// TIA Portal V15.1 export
// export: Created 2024-05-17T05:38:33.8668147Z, ExportSetting WithDefaults, DisplayName Totally Integrated Automation Portal, DisplayVersion V15.1 Update 5, DisplayName TIA Portal Openness, DisplayVersion V15.1 Update 5, DisplayName SINAMICS Startdrive Advanced, DisplayVersion V15.1, DisplayName G130, G150, S120, S150, SINAMICS MV, S210, DisplayVersion V15.1, DisplayName G110M, G120, G120C, G120D, G120P, DisplayVersion V15.1, DisplayName STEP 7 Professional, DisplayVersion V15.1 Update 5, DisplayName STEP 7 Safety, DisplayVersion V15.1, DisplayName WinCC Professional, DisplayVersion V15.1 Update 5, DisplayName SIMATIC Visualization Architect, DisplayVersion V15.1
FUNCTION_BLOCK "LProcSel5SPResFreq"   // FB1733, FBD
TITLE = LProcSel5SPResFreq
{ S7_Optimized_Access := 'FALSE' }
AUTHOR : VCC
FAMILY : ProcEq
NAME : Sel5SP
VERSION : 0.1
// ================================================================================
// This makes the selection of one set-point among 5 in function of the production 
// modes.
// The selection is made via a set-point request integer from 1 to 5.
// An external value is possible to be selected to set-point 1.
// It includes also 5 set-points to reject resonance frequencies if there are.
// ================================================================================
// stored: AutoNumber false, IsIECCheckEnabled false, SetENOAutomatically False, UDAEnableTagReadback false
   VAR_INPUT
      I_ExtSP1_Value { ExternalAccessible := 'False'; ExternalVisible := 'False'; ExternalWritable := 'False'} : Real;   // External Set-point 1
      H_Normalbandwidthmode { ExternalAccessible := 'False'; ExternalVisible := 'False'; ExternalWritable := 'False'} : Bool := TRUE;   // Each resonance frequency his own bandwidth
      H_SPResonance1 : Real;   // Set-point 1 Resonance frequency
      H_SPResonance2 : Real;   // Set-point 2 Resonance frequency
      H_SPResonance3 : Real;   // Set-point 3 Resonance frequency
      H_SPResonance4 : Real;   // Set-point 4 Resonance frequency
      H_SPBandwidth1 : Real;   // Set-point 1 Bandwidth (for resonance frequency)
      H_SPBandwidth2 : Real;   // Set-point 2 Bandwidth (for resonance frequency)
      H_SPBandwidth3 : Real;   // Set-point 3 Bandwidth (for resonance frequency)
      H_SPBandwidth4 : Real;   // Set-point 4 Bandwidth (for resonance frequency)
      I_SPReq : Int;   // Index Set-point Request
      I_ExtSP1 : Bool;   // External Set-point 1 Request
   END_VAR
   VAR_OUTPUT
      O_SPSel : Real;   // Set-point selected
      H_Anim : Word;   // HMI Animation word
   END_VAR
   VAR_IN_OUT
      H_SetpntAllowed : Bool := TRUE;   // Setpoint is OK and allowed
      H_SP1 : Real;   // Set-point 1
      H_SP2 : Real;   // Set-point 2
      H_SP3 : Real;   // Set-point 3
      H_SP4 : Real;   // Set-point 4
      H_SP5 : Real;   // Set-point 5
   END_VAR
   VAR DB_SPECIFIC
      RunNormalOnce { ExternalAccessible := 'False'; ExternalVisible := 'False'; ExternalWritable := 'False'} : Bool := TRUE;   // Check all frequences once - mode is changed
      RunNotNormalOnce { ExternalAccessible := 'False'; ExternalVisible := 'False'; ExternalWritable := 'False'} : Bool;   // Check all frequences once - mode is changed
      SetpntChanged { ExternalAccessible := 'False'; ExternalVisible := 'False'; ExternalWritable := 'False'} : Bool;   // Setpoint is changed
      SetpntResChanged { ExternalAccessible := 'False'; ExternalVisible := 'False'; ExternalWritable := 'False'} : Bool;   // Setpoint Resonance frequency is changed
      SetpntBwdChanged { ExternalAccessible := 'False'; ExternalVisible := 'False'; ExternalWritable := 'False'} : Bool;   // Setpoint bandwidth is changed
      CheckResSetpoints { ExternalAccessible := 'False'; ExternalVisible := 'False'; ExternalWritable := 'False'} : Bool;   // Check all frequences because mode is changed
      ClrGreatestbandwidth { ExternalAccessible := 'False'; ExternalVisible := 'False'; ExternalWritable := 'False'} : Bool;   // Clear greatest bandwidth to search new value
      Greatestbandwidth { ExternalAccessible := 'False'; ExternalVisible := 'False'; ExternalWritable := 'False'} : Real;   // Greatest bandwidth from those who where entered
      MinResSetp1 { ExternalAccessible := 'False'; ExternalVisible := 'False'; ExternalWritable := 'False'} : Real;   // Calculated min. res. Setpoint 1
      MaxResSetp1 { ExternalAccessible := 'False'; ExternalVisible := 'False'; ExternalWritable := 'False'} : Real;   // Calculated max. res. Setpoint 1
      MinResSetp2 { ExternalAccessible := 'False'; ExternalVisible := 'False'; ExternalWritable := 'False'} : Real;   // Calculated min. res. Setpoint 2
      MaxResSetp2 { ExternalAccessible := 'False'; ExternalVisible := 'False'; ExternalWritable := 'False'} : Real;   // Calculated max. res. Setpoint 2
      MinResSetp3 { ExternalAccessible := 'False'; ExternalVisible := 'False'; ExternalWritable := 'False'} : Real;   // Calculated min. res. Setpoint 3
      MaxResSetp3 { ExternalAccessible := 'False'; ExternalVisible := 'False'; ExternalWritable := 'False'} : Real;   // Calculated max. res. Setpoint 3
      MinResSetp4 { ExternalAccessible := 'False'; ExternalVisible := 'False'; ExternalWritable := 'False'} : Real;   // Calculated min. res. Setpoint 4
      MaxResSetp4 { ExternalAccessible := 'False'; ExternalVisible := 'False'; ExternalWritable := 'False'} : Real;   // Calculated max. res. Setpoint 4
      S_NormalBndWdth { ExternalAccessible := 'False'; ExternalVisible := 'False'; ExternalWritable := 'False'} : Bool;   // Step Normal Bandwidth
      S_NoNormalBndWdth { ExternalAccessible := 'False'; ExternalVisible := 'False'; ExternalWritable := 'False'} : Bool;   // Step No Normal Bandwidth
      SPOld1 { ExternalAccessible := 'False'; ExternalVisible := 'False'; ExternalWritable := 'False'} : Real;   // Set-point 1
      SPOld2 { ExternalAccessible := 'False'; ExternalVisible := 'False'; ExternalWritable := 'False'} : Real;   // Set-point 2
      SPOld3 { ExternalAccessible := 'False'; ExternalVisible := 'False'; ExternalWritable := 'False'} : Real;   // Set-point 3
      SPOld4 { ExternalAccessible := 'False'; ExternalVisible := 'False'; ExternalWritable := 'False'} : Real;   // Set-point 4
      SPOld5 { ExternalAccessible := 'False'; ExternalVisible := 'False'; ExternalWritable := 'False'} : Real;   // Set-point 5
      SPResonanceOld1 { ExternalAccessible := 'False'; ExternalVisible := 'False'; ExternalWritable := 'False'} : Real;   // Set-point 1 Resonance frequency
      SPResonanceOld2 { ExternalAccessible := 'False'; ExternalVisible := 'False'; ExternalWritable := 'False'} : Real;   // Set-point 2 Resonance frequency
      SPResonanceOld3 { ExternalAccessible := 'False'; ExternalVisible := 'False'; ExternalWritable := 'False'} : Real;   // Set-point 3 Resonance frequency
      SPResonanceOld4 { ExternalAccessible := 'False'; ExternalVisible := 'False'; ExternalWritable := 'False'} : Real;   // Set-point 4 Resonance frequency
      SPBandwidthOld1 { ExternalAccessible := 'False'; ExternalVisible := 'False'; ExternalWritable := 'False'} : Real;   // Set-point 1 Bandwidth (for resonance frequency)
      SPBandwidthOld2 { ExternalAccessible := 'False'; ExternalVisible := 'False'; ExternalWritable := 'False'} : Real;   // Set-point 2 Bandwidth (for resonance frequency)
      SPBandwidthOld3 { ExternalAccessible := 'False'; ExternalVisible := 'False'; ExternalWritable := 'False'} : Real;   // Set-point 3 Bandwidth (for resonance frequency)
      SPBandwidthOld4 { ExternalAccessible := 'False'; ExternalVisible := 'False'; ExternalWritable := 'False'} : Real;   // Set-point 4 Bandwidth (for resonance frequency)
   END_VAR
   VAR_TEMP   // added for the SCL form of the ladder/FBD networks
      _w1 : Bool;
      _w2 : Bool;
      _w3 : Bool;
   END_VAR
BEGIN

REGION Network 1: **** 4.6 - Machine status - Indications **** Controller Animation word 1 for HMI
   // Controller Animation word 1 for HMI
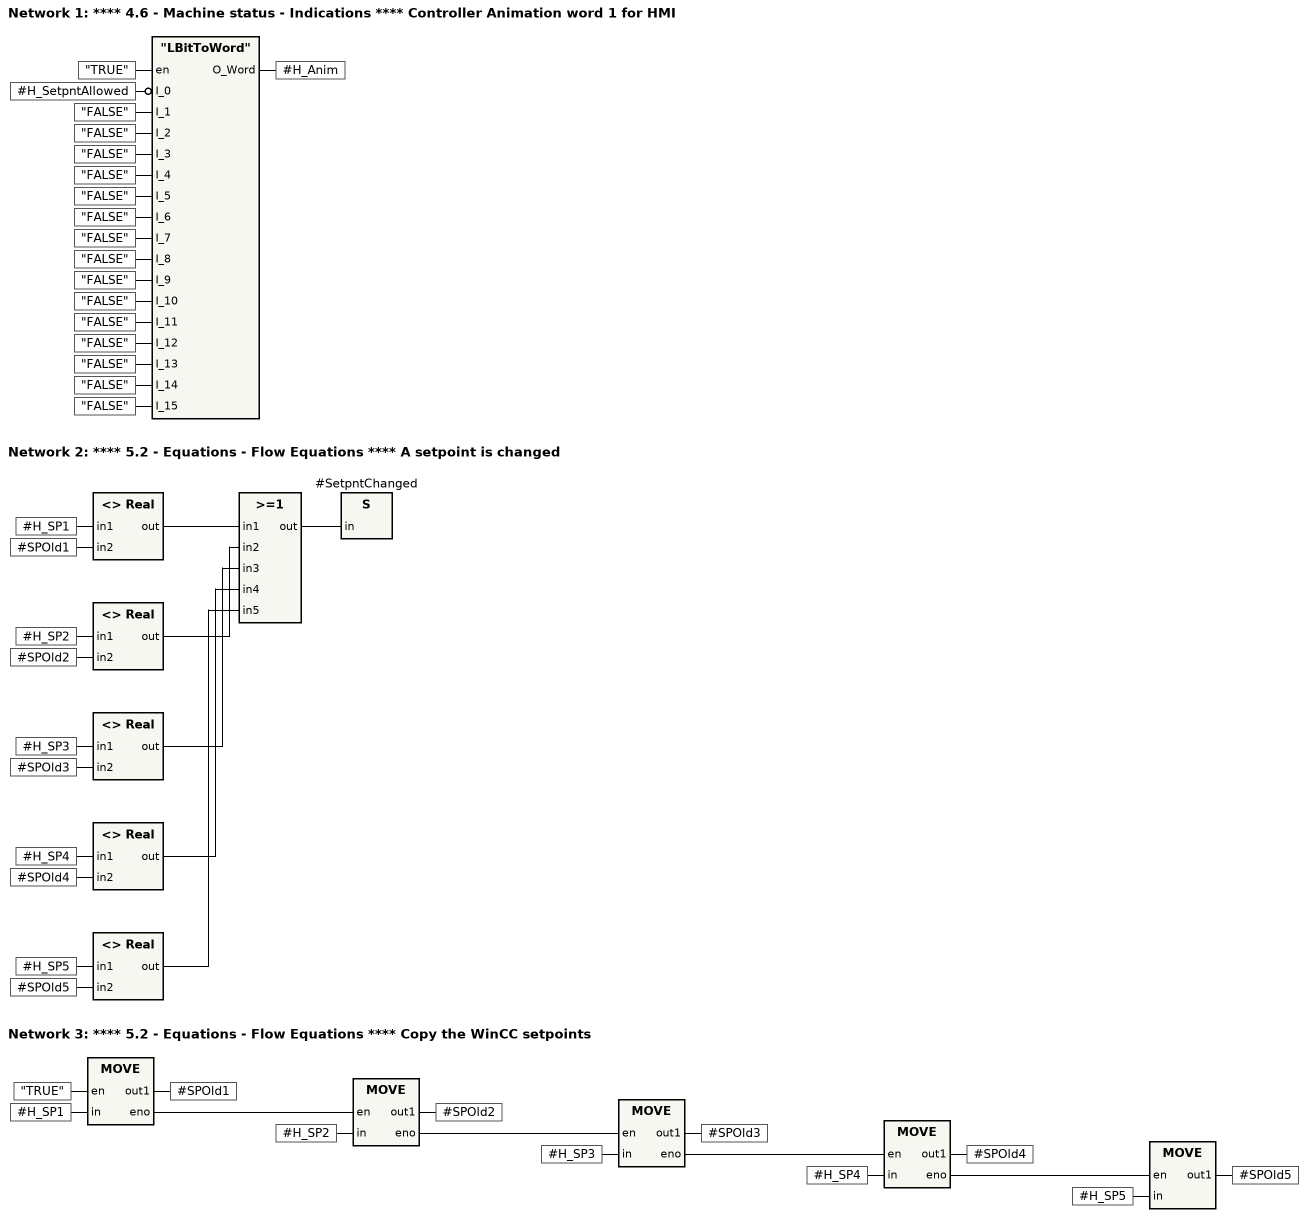
   IF "TRUE" THEN
       "LBitToWord"(I_0 := NOT #H_SetpntAllowed,
                    I_1 := "FALSE",
                    I_2 := "FALSE",
                    I_3 := "FALSE",
                    I_4 := "FALSE",
                    I_5 := "FALSE",
                    I_6 := "FALSE",
                    I_7 := "FALSE",
                    I_8 := "FALSE",
                    I_9 := "FALSE",
                    I_10 := "FALSE",
                    I_11 := "FALSE",
                    I_12 := "FALSE",
                    I_13 := "FALSE",
                    I_14 := "FALSE",
                    I_15 := "FALSE",
                    O_Word => #H_Anim);
   END_IF;
END_REGION

REGION Network 2: **** 5.2 - Equations - Flow Equations **** A setpoint is changed
   // A setpoint is changed
   IF (#H_SP1 <> #SPOld1) OR (#H_SP2 <> #SPOld2) OR (#H_SP3 <> #SPOld3) OR (#H_SP4 <> #SPOld4) OR (#H_SP5 <> #SPOld5) THEN
       #SetpntChanged := TRUE;
   END_IF;
END_REGION

REGION Network 3: **** 5.2 - Equations - Flow Equations **** Copy the WinCC setpoints
   // Copy the WinCC setpoints
   // ENO of a box is taken as its EN; it also drops when the box reports an error
   IF "TRUE" THEN
       #SPOld1 := #H_SP1;
       #SPOld2 := #H_SP2;
       #SPOld3 := #H_SP3;
       #SPOld4 := #H_SP4;
       #SPOld5 := #H_SP5;
   END_IF;
END_REGION

REGION Network 4: **** 5.2 - Equations - Flow Equations **** A setpoint of resonance is changed
   // A setpoint of resonance is changed
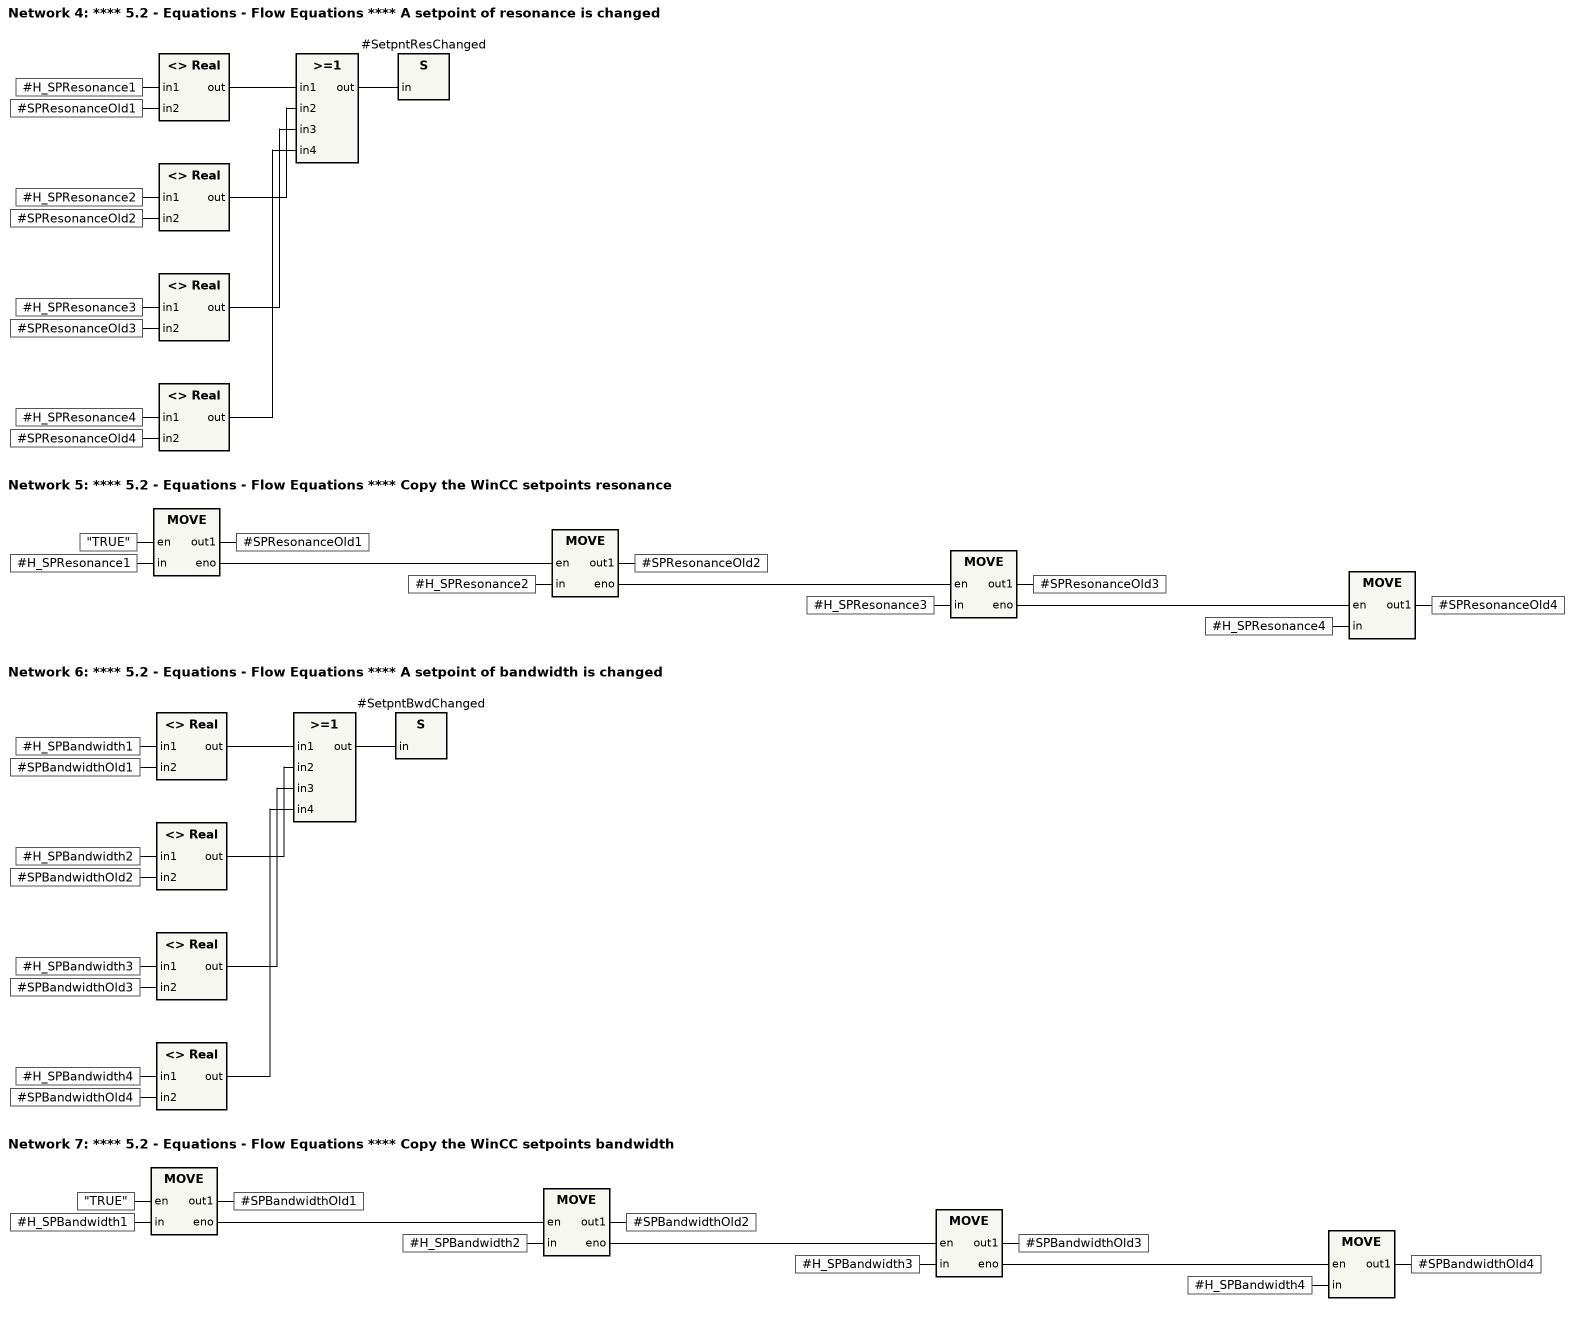
   IF (#H_SPResonance1 <> #SPResonanceOld1) OR (#H_SPResonance2 <> #SPResonanceOld2) OR (#H_SPResonance3 <> #SPResonanceOld3) OR (#H_SPResonance4 <> #SPResonanceOld4) THEN
       #SetpntResChanged := TRUE;
   END_IF;
END_REGION

REGION Network 5: **** 5.2 - Equations - Flow Equations **** Copy the WinCC setpoints resonance
   // Copy the WinCC setpoints resonance
   // ENO of a box is taken as its EN; it also drops when the box reports an error
   IF "TRUE" THEN
       #SPResonanceOld1 := #H_SPResonance1;
       #SPResonanceOld2 := #H_SPResonance2;
       #SPResonanceOld3 := #H_SPResonance3;
       #SPResonanceOld4 := #H_SPResonance4;
   END_IF;
END_REGION

REGION Network 6: **** 5.2 - Equations - Flow Equations **** A setpoint of bandwidth is changed
   // A setpoint of bandwidth is changed
   IF (#H_SPBandwidth1 <> #SPBandwidthOld1) OR (#H_SPBandwidth2 <> #SPBandwidthOld2) OR (#H_SPBandwidth3 <> #SPBandwidthOld3) OR (#H_SPBandwidth4 <> #SPBandwidthOld4) THEN
       #SetpntBwdChanged := TRUE;
   END_IF;
END_REGION

REGION Network 7: **** 5.2 - Equations - Flow Equations **** Copy the WinCC setpoints bandwidth
   // Copy the WinCC setpoints bandwidth
   // ENO of a box is taken as its EN; it also drops when the box reports an error
   IF "TRUE" THEN
       #SPBandwidthOld1 := #H_SPBandwidth1;
       #SPBandwidthOld2 := #H_SPBandwidth2;
       #SPBandwidthOld3 := #H_SPBandwidth3;
       #SPBandwidthOld4 := #H_SPBandwidth4;
   END_IF;
END_REGION

REGION Network 8: **** 5.2 - Equations - Flow Equations **** Selection Set-point 1
   // Selection Set-point 1
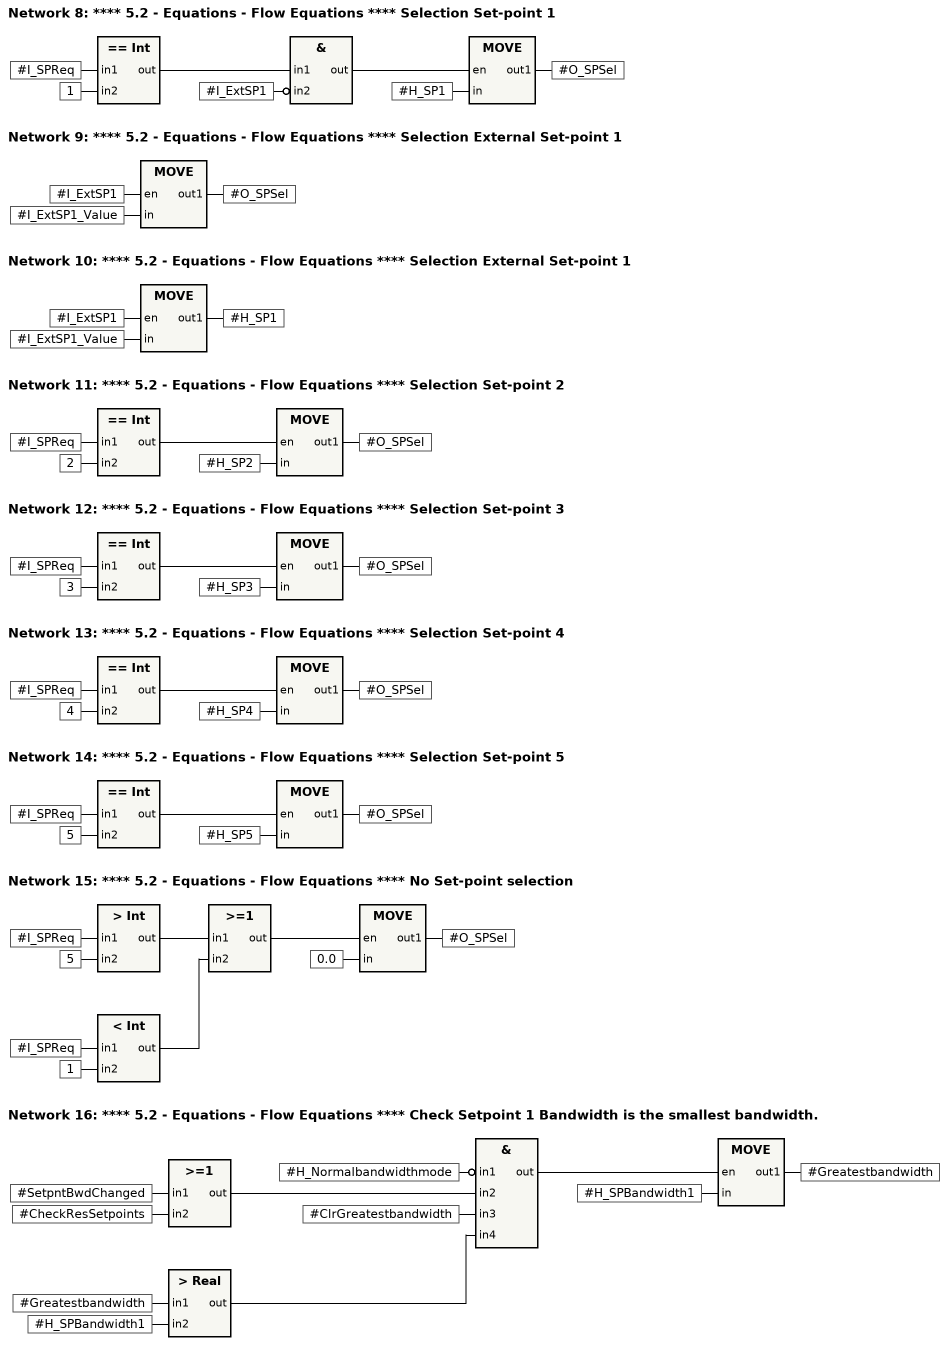
   IF (#I_SPReq = 1) AND NOT #I_ExtSP1 THEN #O_SPSel := #H_SP1; END_IF;
END_REGION

REGION Network 9: **** 5.2 - Equations - Flow Equations **** Selection External Set-point 1
   // Selection External Set-point 1
   IF #I_ExtSP1 THEN #O_SPSel := #I_ExtSP1_Value; END_IF;
END_REGION

REGION Network 10: **** 5.2 - Equations - Flow Equations **** Selection External Set-point 1
   // Selection External Set-point 1
   IF #I_ExtSP1 THEN #H_SP1 := #I_ExtSP1_Value; END_IF;
END_REGION

REGION Network 11: **** 5.2 - Equations - Flow Equations **** Selection Set-point 2
   // Selection Set-point 2
   IF #I_SPReq = 2 THEN #O_SPSel := #H_SP2; END_IF;
END_REGION

REGION Network 12: **** 5.2 - Equations - Flow Equations **** Selection Set-point 3
   // Selection Set-point 3
   IF #I_SPReq = 3 THEN #O_SPSel := #H_SP3; END_IF;
END_REGION

REGION Network 13: **** 5.2 - Equations - Flow Equations **** Selection Set-point 4
   // Selection Set-point 4
   IF #I_SPReq = 4 THEN #O_SPSel := #H_SP4; END_IF;
END_REGION

REGION Network 14: **** 5.2 - Equations - Flow Equations **** Selection Set-point 5
   // Selection Set-point 5
   IF #I_SPReq = 5 THEN #O_SPSel := #H_SP5; END_IF;
END_REGION

REGION Network 15: **** 5.2 - Equations - Flow Equations **** No Set-point selection
   // No Set-point selection
   IF (#I_SPReq > 5) OR (#I_SPReq < 1) THEN #O_SPSel := 0.0; END_IF;
END_REGION

REGION Network 16: **** 5.2 - Equations - Flow Equations **** Check Setpoint 1 Bandwidth is the smallest bandwidth.
   // Check Setpoint 1 Bandwidth is the smallest bandwidth.
   IF NOT #H_Normalbandwidthmode AND (#SetpntBwdChanged OR #CheckResSetpoints) AND #ClrGreatestbandwidth AND (#Greatestbandwidth > #H_SPBandwidth1) THEN
       #Greatestbandwidth := #H_SPBandwidth1;
   END_IF;
END_REGION

REGION Network 17: **** 5.2 - Equations - Flow Equations **** Check Setpoint 2 Bandwidth is the smallest bandwidth.
   // Check Setpoint 2 Bandwidth is the smallest bandwidth.
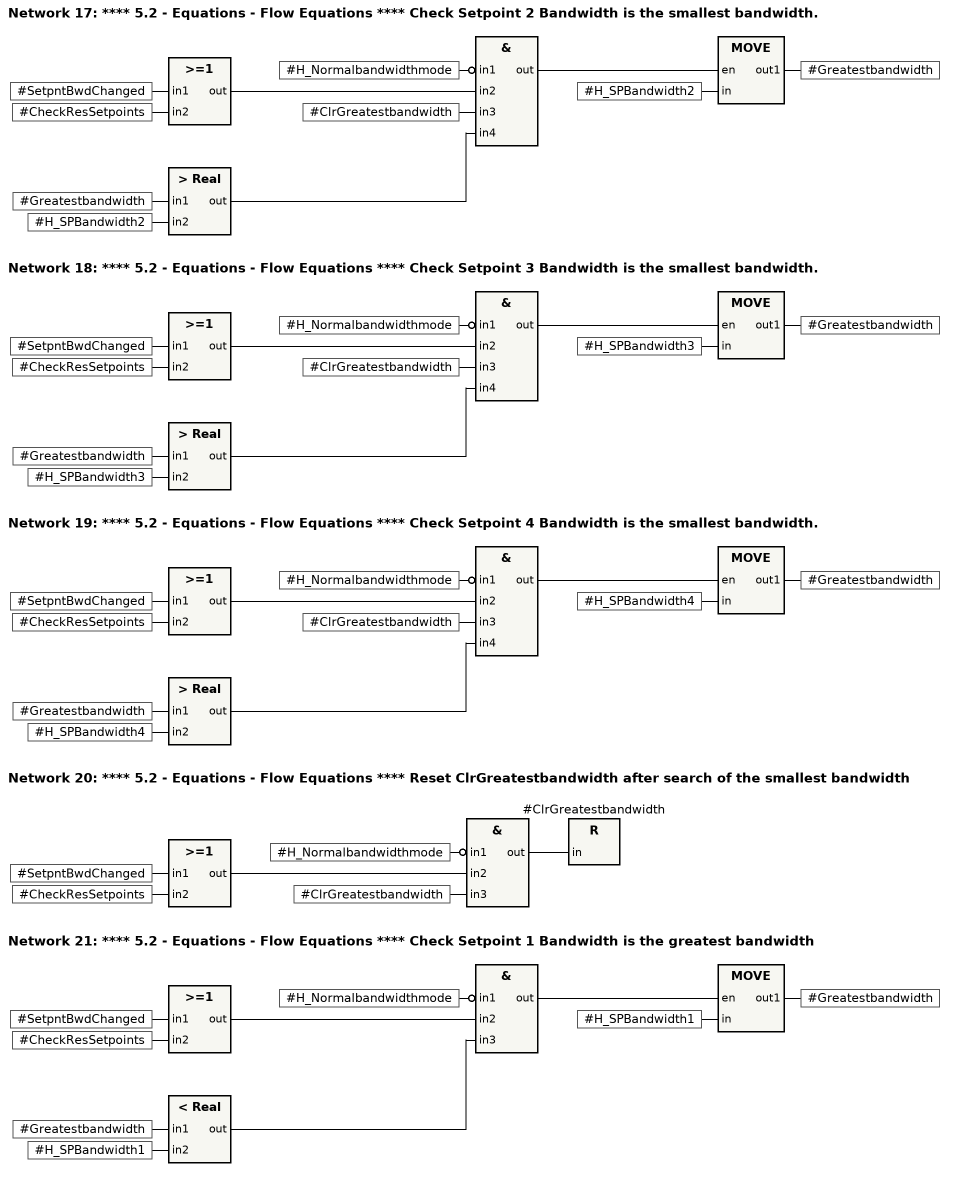
   IF NOT #H_Normalbandwidthmode AND (#SetpntBwdChanged OR #CheckResSetpoints) AND #ClrGreatestbandwidth AND (#Greatestbandwidth > #H_SPBandwidth2) THEN
       #Greatestbandwidth := #H_SPBandwidth2;
   END_IF;
END_REGION

REGION Network 18: **** 5.2 - Equations - Flow Equations **** Check Setpoint 3 Bandwidth is the smallest bandwidth.
   // Check Setpoint 3 Bandwidth is the smallest bandwidth.
   IF NOT #H_Normalbandwidthmode AND (#SetpntBwdChanged OR #CheckResSetpoints) AND #ClrGreatestbandwidth AND (#Greatestbandwidth > #H_SPBandwidth3) THEN
       #Greatestbandwidth := #H_SPBandwidth3;
   END_IF;
END_REGION

REGION Network 19: **** 5.2 - Equations - Flow Equations **** Check Setpoint 4 Bandwidth is the smallest bandwidth.
   // Check Setpoint 4 Bandwidth is the smallest bandwidth.
   IF NOT #H_Normalbandwidthmode AND (#SetpntBwdChanged OR #CheckResSetpoints) AND #ClrGreatestbandwidth AND (#Greatestbandwidth > #H_SPBandwidth4) THEN
       #Greatestbandwidth := #H_SPBandwidth4;
   END_IF;
END_REGION

REGION Network 20: **** 5.2 - Equations - Flow Equations **** Reset ClrGreatestbandwidth after search of the smallest bandwidth
   // Reset ClrGreatestbandwidth after search of the smallest bandwidth
   IF NOT #H_Normalbandwidthmode AND (#SetpntBwdChanged OR #CheckResSetpoints) AND #ClrGreatestbandwidth THEN
       #ClrGreatestbandwidth := FALSE;
   END_IF;
END_REGION

REGION Network 21: **** 5.2 - Equations - Flow Equations **** Check Setpoint 1 Bandwidth is the greatest bandwidth
   // Check Setpoint 1 Bandwidth is the greatest bandwidth
   IF NOT #H_Normalbandwidthmode AND (#SetpntBwdChanged OR #CheckResSetpoints) AND (#Greatestbandwidth < #H_SPBandwidth1) THEN
       #Greatestbandwidth := #H_SPBandwidth1;
   END_IF;
END_REGION

REGION Network 22: **** 5.2 - Equations - Flow Equations **** Check Setpoint 2 Bandwidth is the greatest bandwidth
   // Check Setpoint 2 Bandwidth is the greatest bandwidth
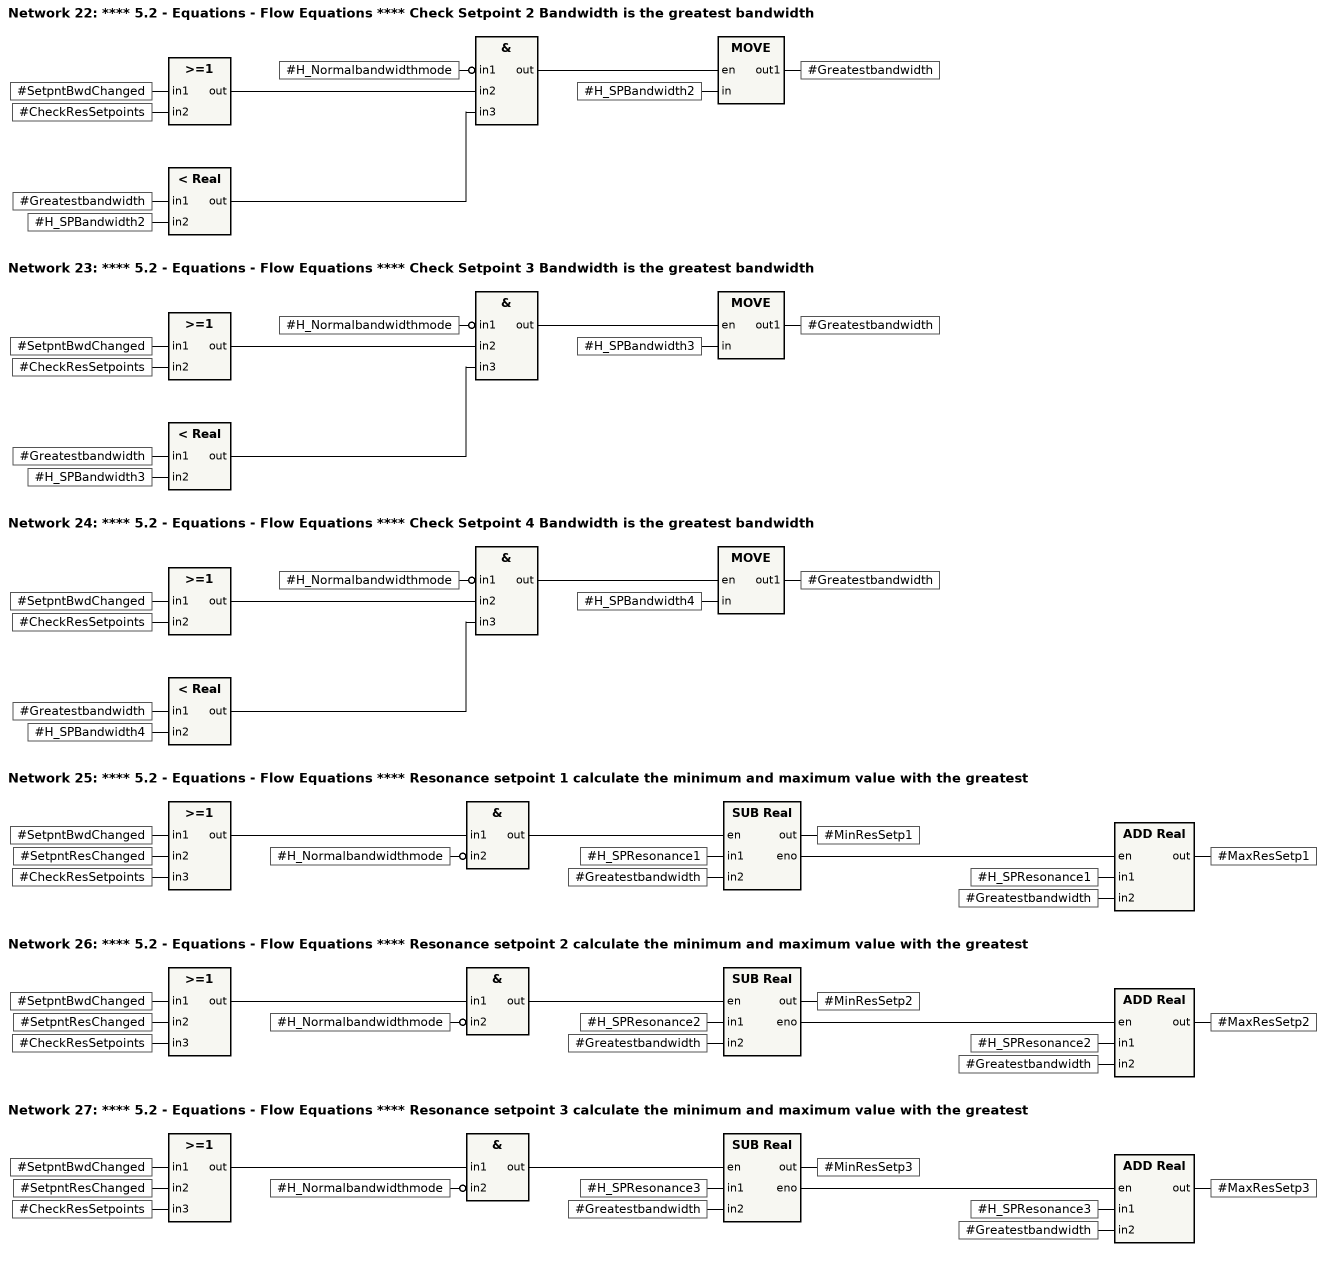
   IF NOT #H_Normalbandwidthmode AND (#SetpntBwdChanged OR #CheckResSetpoints) AND (#Greatestbandwidth < #H_SPBandwidth2) THEN
       #Greatestbandwidth := #H_SPBandwidth2;
   END_IF;
END_REGION

REGION Network 23: **** 5.2 - Equations - Flow Equations **** Check Setpoint 3 Bandwidth is the greatest bandwidth
   // Check Setpoint 3 Bandwidth is the greatest bandwidth
   IF NOT #H_Normalbandwidthmode AND (#SetpntBwdChanged OR #CheckResSetpoints) AND (#Greatestbandwidth < #H_SPBandwidth3) THEN
       #Greatestbandwidth := #H_SPBandwidth3;
   END_IF;
END_REGION

REGION Network 24: **** 5.2 - Equations - Flow Equations **** Check Setpoint 4 Bandwidth is the greatest bandwidth
   // Check Setpoint 4 Bandwidth is the greatest bandwidth
   IF NOT #H_Normalbandwidthmode AND (#SetpntBwdChanged OR #CheckResSetpoints) AND (#Greatestbandwidth < #H_SPBandwidth4) THEN
       #Greatestbandwidth := #H_SPBandwidth4;
   END_IF;
END_REGION

REGION Network 25: **** 5.2 - Equations - Flow Equations **** Resonance setpoint 1 calculate the minimum and maximum value with the greatest
   // Resonance setpoint 1 calculate the minimum and maximum value with the greatest 
   // bandwidth
   // ENO of a box is taken as its EN; it also drops when the box reports an error
   IF (#SetpntBwdChanged OR #SetpntResChanged OR #CheckResSetpoints) AND NOT #H_Normalbandwidthmode THEN
       #MinResSetp1 := #H_SPResonance1 - #Greatestbandwidth;
       #MaxResSetp1 := #H_SPResonance1 + #Greatestbandwidth;
   END_IF;
END_REGION

REGION Network 26: **** 5.2 - Equations - Flow Equations **** Resonance setpoint 2 calculate the minimum and maximum value with the greatest
   // Resonance setpoint 2 calculate the minimum and maximum value with the greatest 
   // bandwidth
   // ENO of a box is taken as its EN; it also drops when the box reports an error
   IF (#SetpntBwdChanged OR #SetpntResChanged OR #CheckResSetpoints) AND NOT #H_Normalbandwidthmode THEN
       #MinResSetp2 := #H_SPResonance2 - #Greatestbandwidth;
       #MaxResSetp2 := #H_SPResonance2 + #Greatestbandwidth;
   END_IF;
END_REGION

REGION Network 27: **** 5.2 - Equations - Flow Equations **** Resonance setpoint 3 calculate the minimum and maximum value with the greatest
   // Resonance setpoint 3 calculate the minimum and maximum value with the greatest 
   // bandwidth
   // ENO of a box is taken as its EN; it also drops when the box reports an error
   IF (#SetpntBwdChanged OR #SetpntResChanged OR #CheckResSetpoints) AND NOT #H_Normalbandwidthmode THEN
       #MinResSetp3 := #H_SPResonance3 - #Greatestbandwidth;
       #MaxResSetp3 := #H_SPResonance3 + #Greatestbandwidth;
   END_IF;
END_REGION

REGION Network 28: **** 5.2 - Equations - Flow Equations **** Resonance setpoint 4 calculate the minimum and maximum value with the greatest
   // Resonance setpoint 4 calculate the minimum and maximum value with the greatest 
   // bandwidth
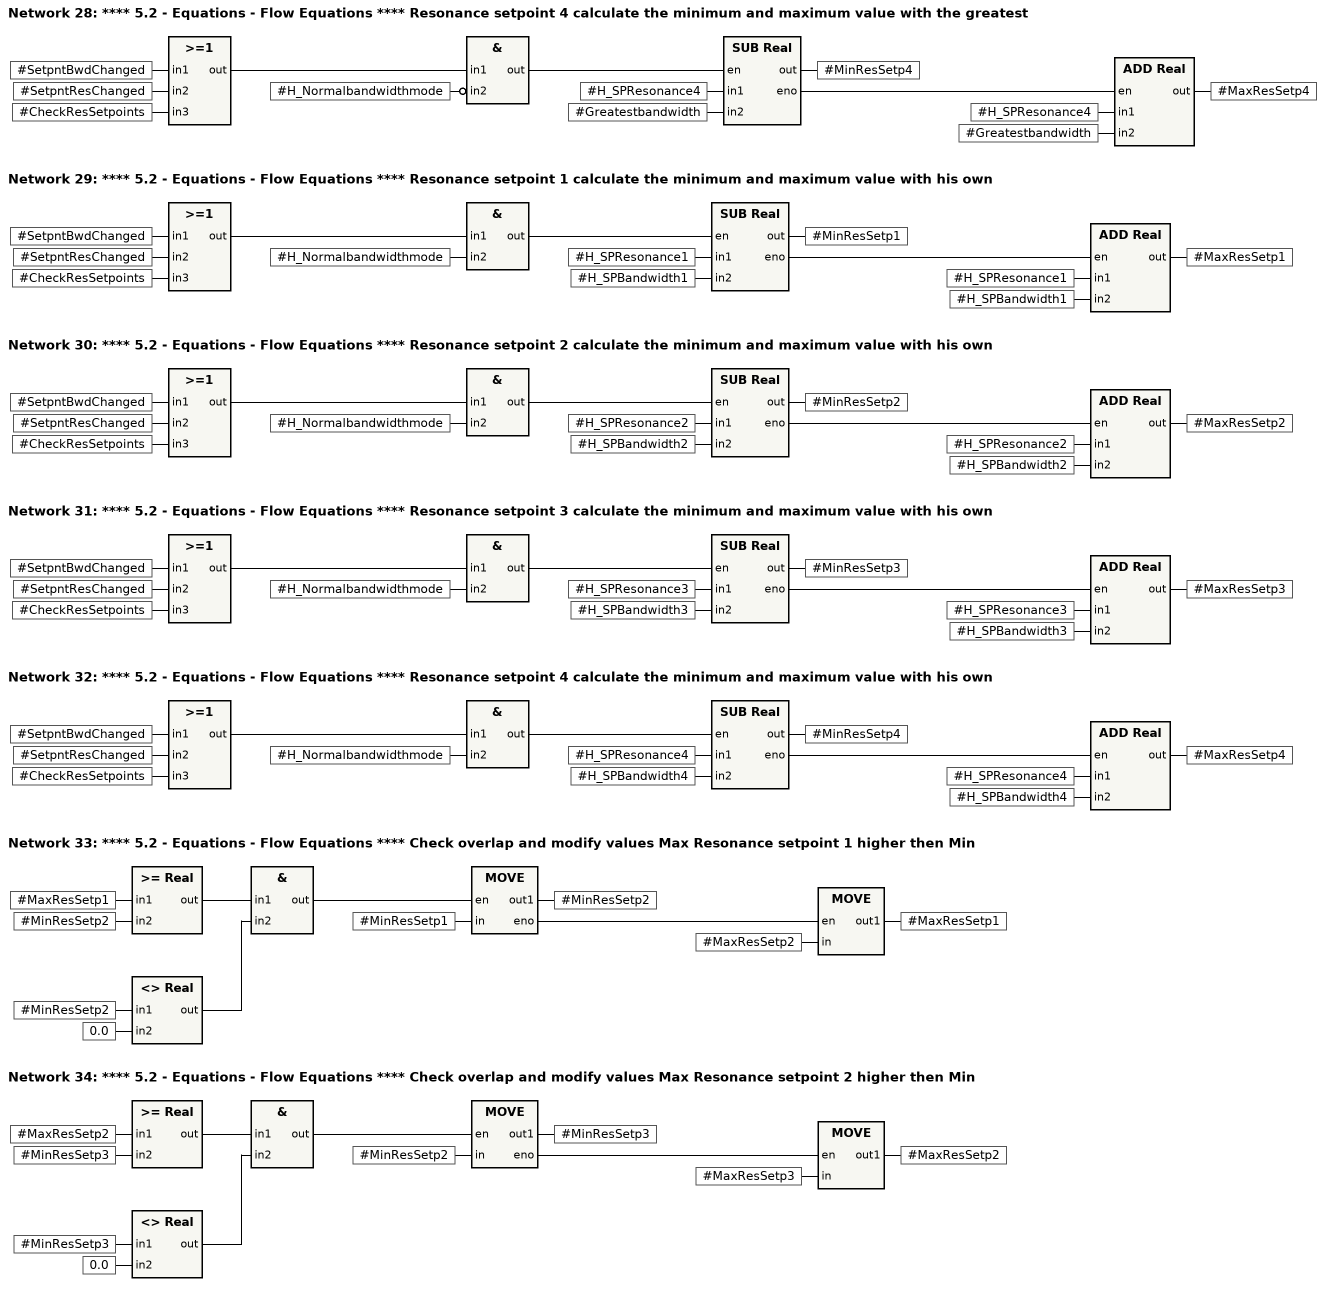
   // ENO of a box is taken as its EN; it also drops when the box reports an error
   IF (#SetpntBwdChanged OR #SetpntResChanged OR #CheckResSetpoints) AND NOT #H_Normalbandwidthmode THEN
       #MinResSetp4 := #H_SPResonance4 - #Greatestbandwidth;
       #MaxResSetp4 := #H_SPResonance4 + #Greatestbandwidth;
   END_IF;
END_REGION

REGION Network 29: **** 5.2 - Equations - Flow Equations **** Resonance setpoint 1 calculate the minimum and maximum value with his own
   // Resonance setpoint 1 calculate the minimum and maximum value with his own 
   // bandwidth
   // ENO of a box is taken as its EN; it also drops when the box reports an error
   IF (#SetpntBwdChanged OR #SetpntResChanged OR #CheckResSetpoints) AND #H_Normalbandwidthmode THEN
       #MinResSetp1 := #H_SPResonance1 - #H_SPBandwidth1;
       #MaxResSetp1 := #H_SPResonance1 + #H_SPBandwidth1;
   END_IF;
END_REGION

REGION Network 30: **** 5.2 - Equations - Flow Equations **** Resonance setpoint 2 calculate the minimum and maximum value with his own
   // Resonance setpoint 2 calculate the minimum and maximum value with his own 
   // bandwidth
   // ENO of a box is taken as its EN; it also drops when the box reports an error
   IF (#SetpntBwdChanged OR #SetpntResChanged OR #CheckResSetpoints) AND #H_Normalbandwidthmode THEN
       #MinResSetp2 := #H_SPResonance2 - #H_SPBandwidth2;
       #MaxResSetp2 := #H_SPResonance2 + #H_SPBandwidth2;
   END_IF;
END_REGION

REGION Network 31: **** 5.2 - Equations - Flow Equations **** Resonance setpoint 3 calculate the minimum and maximum value with his own
   // Resonance setpoint 3 calculate the minimum and maximum value with his own 
   // bandwidth
   // ENO of a box is taken as its EN; it also drops when the box reports an error
   IF (#SetpntBwdChanged OR #SetpntResChanged OR #CheckResSetpoints) AND #H_Normalbandwidthmode THEN
       #MinResSetp3 := #H_SPResonance3 - #H_SPBandwidth3;
       #MaxResSetp3 := #H_SPResonance3 + #H_SPBandwidth3;
   END_IF;
END_REGION

REGION Network 32: **** 5.2 - Equations - Flow Equations **** Resonance setpoint 4 calculate the minimum and maximum value with his own
   // Resonance setpoint 4 calculate the minimum and maximum value with his own 
   // bandwidth
   // ENO of a box is taken as its EN; it also drops when the box reports an error
   IF (#SetpntBwdChanged OR #SetpntResChanged OR #CheckResSetpoints) AND #H_Normalbandwidthmode THEN
       #MinResSetp4 := #H_SPResonance4 - #H_SPBandwidth4;
       #MaxResSetp4 := #H_SPResonance4 + #H_SPBandwidth4;
   END_IF;
END_REGION

REGION Network 33: **** 5.2 - Equations - Flow Equations **** Check overlap and modify values Max Resonance setpoint 1 higher then Min
   // Check overlap and modify values Max Resonance setpoint 1 higher then Min 
   // Resonance setpoint 2
   // ENO of a box is taken as its EN; it also drops when the box reports an error
   #_w1 := (#MaxResSetp1 >= #MinResSetp2) AND (#MinResSetp2 <> 0.0);
   IF #_w1 THEN
       #MinResSetp2 := #MinResSetp1;
       #MaxResSetp1 := #MaxResSetp2;
   END_IF;
END_REGION

REGION Network 34: **** 5.2 - Equations - Flow Equations **** Check overlap and modify values Max Resonance setpoint 2 higher then Min
   // Check overlap and modify values Max Resonance setpoint 2 higher then Min 
   // Resonance setpoint 3
   // ENO of a box is taken as its EN; it also drops when the box reports an error
   #_w1 := (#MaxResSetp2 >= #MinResSetp3) AND (#MinResSetp3 <> 0.0);
   IF #_w1 THEN
       #MinResSetp3 := #MinResSetp2;
       #MaxResSetp2 := #MaxResSetp3;
   END_IF;
END_REGION

REGION Network 35: **** 5.2 - Equations - Flow Equations **** Check overlap and modify values Max Resonance setpoint 3 higher then Min
   // Check overlap and modify values Max Resonance setpoint 3 higher then Min 
   // Resonance setpoint 4
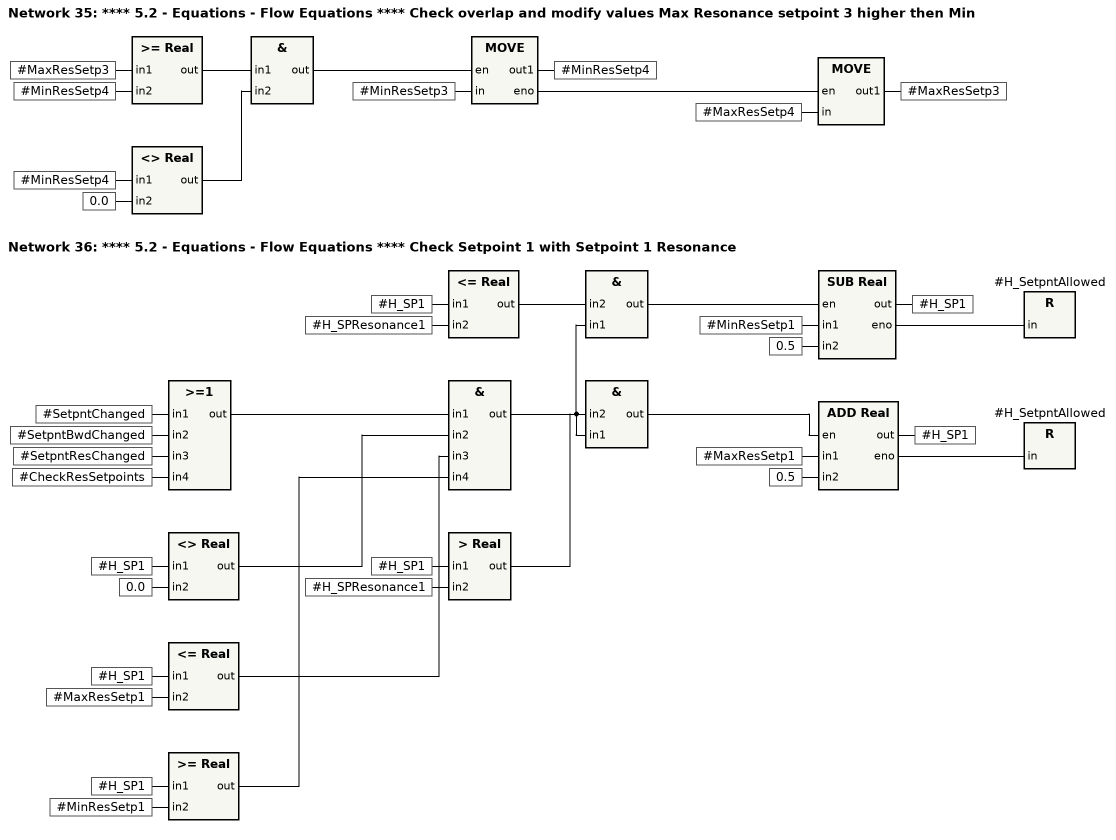
   // ENO of a box is taken as its EN; it also drops when the box reports an error
   #_w1 := (#MaxResSetp3 >= #MinResSetp4) AND (#MinResSetp4 <> 0.0);
   IF #_w1 THEN
       #MinResSetp4 := #MinResSetp3;
       #MaxResSetp3 := #MaxResSetp4;
   END_IF;
END_REGION

REGION Network 36: **** 5.2 - Equations - Flow Equations **** Check Setpoint 1 with Setpoint 1 Resonance
   // Check Setpoint 1 with Setpoint 1 Resonance 
   // Setpoint 1 is no longer allowed, calculate prefered allowed setpoint 1
   // ENO of a box is taken as its EN; it also drops when the box reports an error
   #_w1 := (#SetpntChanged OR #SetpntBwdChanged OR #SetpntResChanged OR #CheckResSetpoints) AND (#H_SP1 <> 0.0) AND (#H_SP1 <= #MaxResSetp1) AND (#H_SP1 >= #MinResSetp1);
   #_w2 := (#H_SP1 <= #H_SPResonance1) AND #_w1;
   IF #_w2 THEN
       #H_SP1 := #MinResSetp1 - 0.5;
       #H_SetpntAllowed := FALSE;
   END_IF;
   #_w3 := (#H_SP1 > #H_SPResonance1) AND #_w1;
   IF #_w3 THEN
       #H_SP1 := #MaxResSetp1 + 0.5;
       #H_SetpntAllowed := FALSE;
   END_IF;
END_REGION

REGION Network 37: **** 5.2 - Equations - Flow Equations **** Check Setpoint 1 with Setpoint 2 Resonance
   // Check Setpoint 1 with Setpoint 2 Resonance 
   // Setpoint 1 is no longer allowed, calculate prefered allowed setpoint 1
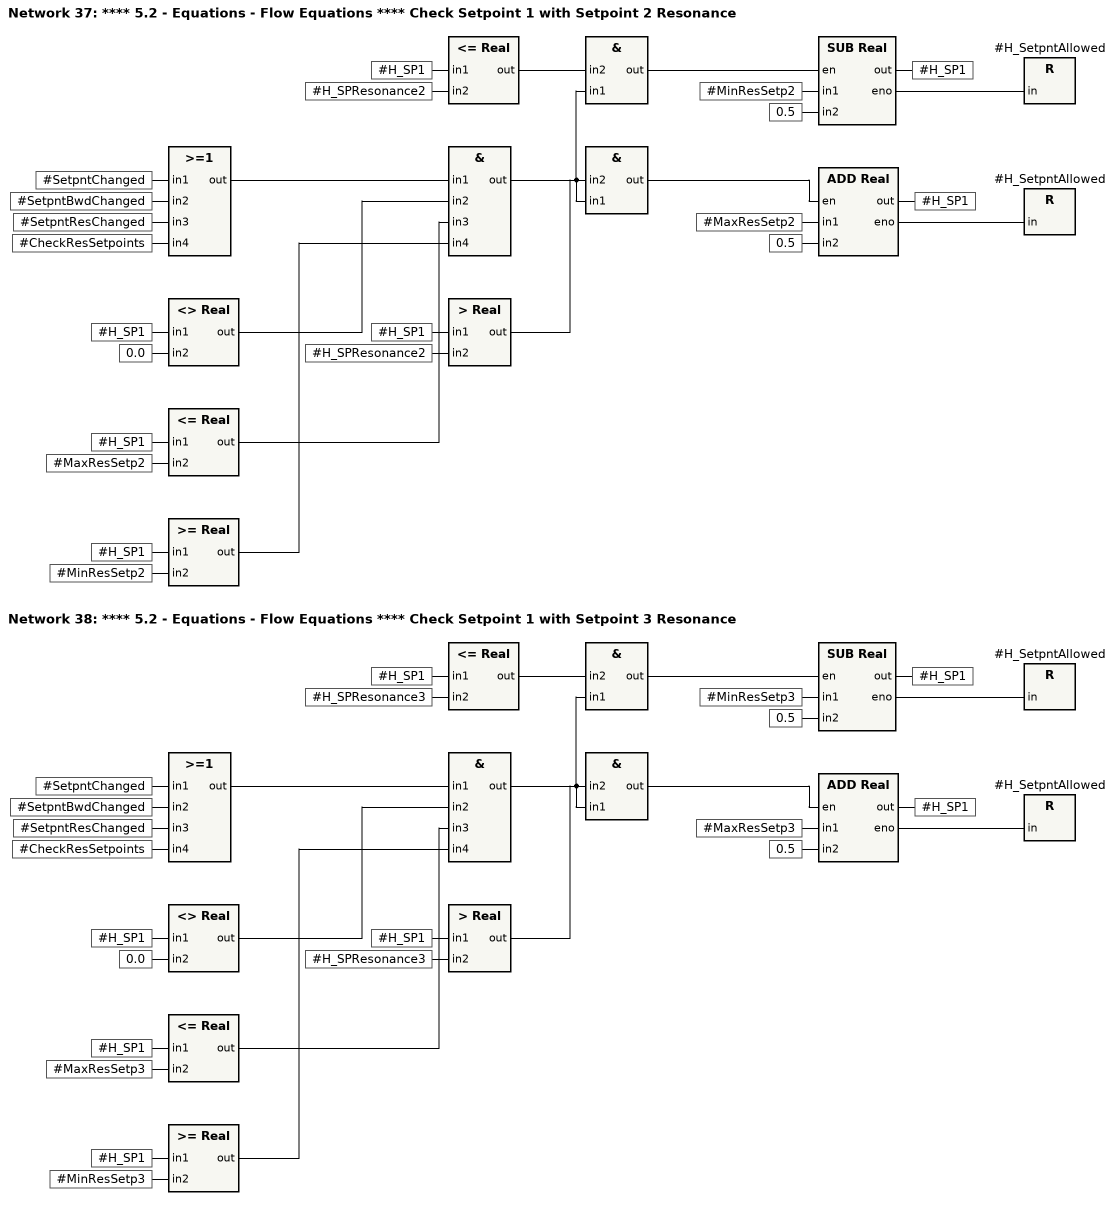
   // ENO of a box is taken as its EN; it also drops when the box reports an error
   #_w1 := (#SetpntChanged OR #SetpntBwdChanged OR #SetpntResChanged OR #CheckResSetpoints) AND (#H_SP1 <> 0.0) AND (#H_SP1 <= #MaxResSetp2) AND (#H_SP1 >= #MinResSetp2);
   #_w2 := (#H_SP1 <= #H_SPResonance2) AND #_w1;
   IF #_w2 THEN
       #H_SP1 := #MinResSetp2 - 0.5;
       #H_SetpntAllowed := FALSE;
   END_IF;
   #_w3 := (#H_SP1 > #H_SPResonance2) AND #_w1;
   IF #_w3 THEN
       #H_SP1 := #MaxResSetp2 + 0.5;
       #H_SetpntAllowed := FALSE;
   END_IF;
END_REGION

REGION Network 38: **** 5.2 - Equations - Flow Equations **** Check Setpoint 1 with Setpoint 3 Resonance
   // Check Setpoint 1 with Setpoint 3 Resonance 
   // Setpoint 1 is no longer allowed, calculate prefered allowed setpoint 1
   // ENO of a box is taken as its EN; it also drops when the box reports an error
   #_w1 := (#SetpntChanged OR #SetpntBwdChanged OR #SetpntResChanged OR #CheckResSetpoints) AND (#H_SP1 <> 0.0) AND (#H_SP1 <= #MaxResSetp3) AND (#H_SP1 >= #MinResSetp3);
   #_w2 := (#H_SP1 <= #H_SPResonance3) AND #_w1;
   IF #_w2 THEN
       #H_SP1 := #MinResSetp3 - 0.5;
       #H_SetpntAllowed := FALSE;
   END_IF;
   #_w3 := (#H_SP1 > #H_SPResonance3) AND #_w1;
   IF #_w3 THEN
       #H_SP1 := #MaxResSetp3 + 0.5;
       #H_SetpntAllowed := FALSE;
   END_IF;
END_REGION

REGION Network 39: **** 5.2 - Equations - Flow Equations **** Check Setpoint 1 with Setpoint 4 Resonance
   // Check Setpoint 1 with Setpoint 4 Resonance 
   // Setpoint 1 is no longer allowed, calculate prefered allowed setpoint 1
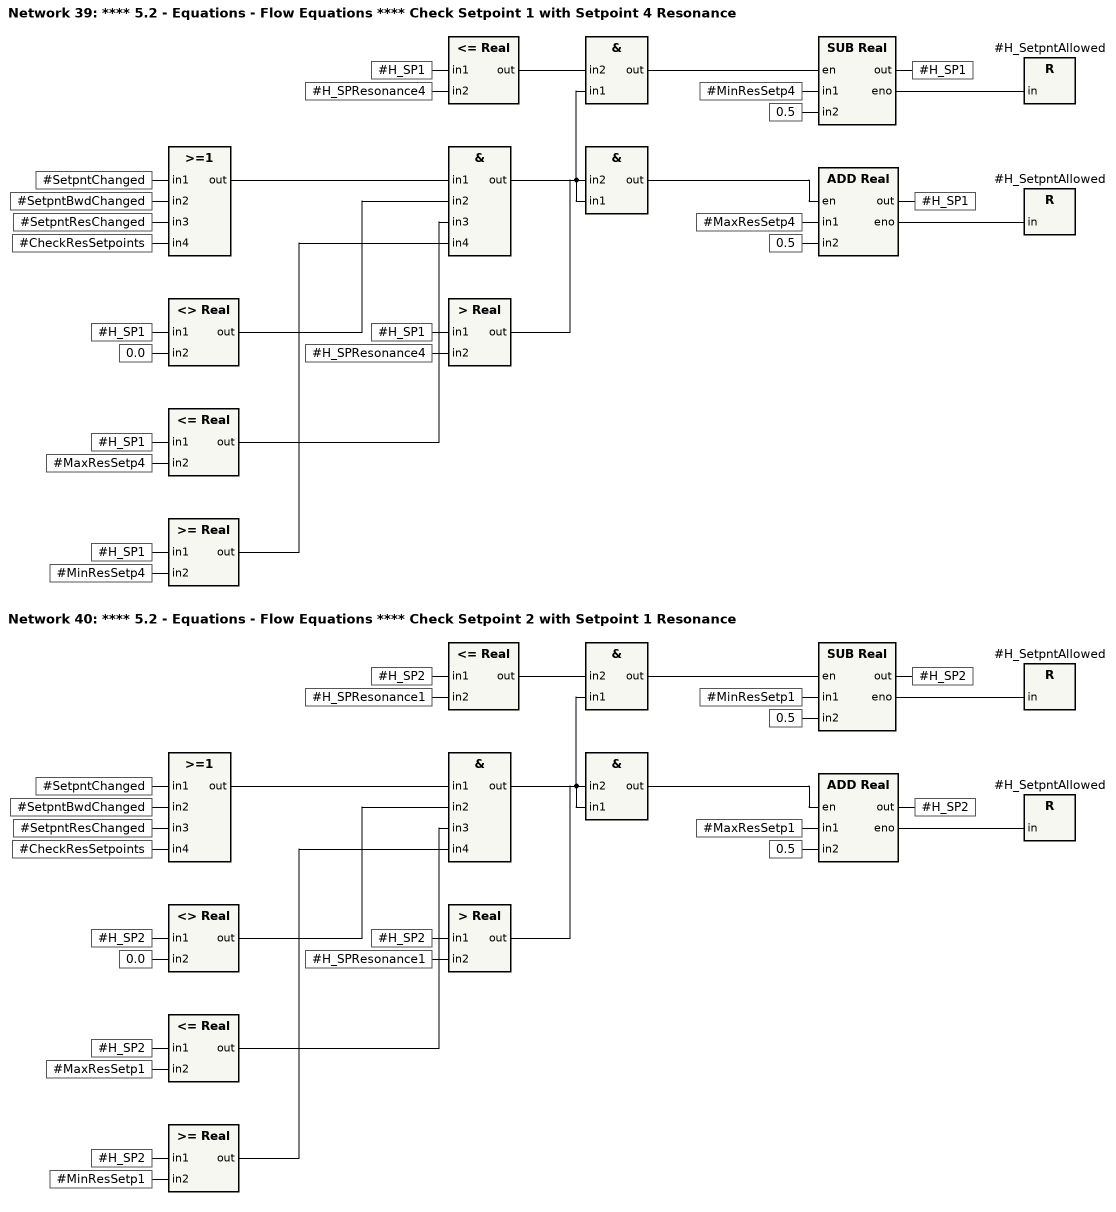
   // ENO of a box is taken as its EN; it also drops when the box reports an error
   #_w1 := (#SetpntChanged OR #SetpntBwdChanged OR #SetpntResChanged OR #CheckResSetpoints) AND (#H_SP1 <> 0.0) AND (#H_SP1 <= #MaxResSetp4) AND (#H_SP1 >= #MinResSetp4);
   #_w2 := (#H_SP1 <= #H_SPResonance4) AND #_w1;
   IF #_w2 THEN
       #H_SP1 := #MinResSetp4 - 0.5;
       #H_SetpntAllowed := FALSE;
   END_IF;
   #_w3 := (#H_SP1 > #H_SPResonance4) AND #_w1;
   IF #_w3 THEN
       #H_SP1 := #MaxResSetp4 + 0.5;
       #H_SetpntAllowed := FALSE;
   END_IF;
END_REGION

REGION Network 40: **** 5.2 - Equations - Flow Equations **** Check Setpoint 2 with Setpoint 1 Resonance
   // Check Setpoint 2 with Setpoint 1 Resonance 
   // Setpoint 2 is no longer allowed, calculate prefered allowed setpoint 2
   // ENO of a box is taken as its EN; it also drops when the box reports an error
   #_w1 := (#SetpntChanged OR #SetpntBwdChanged OR #SetpntResChanged OR #CheckResSetpoints) AND (#H_SP2 <> 0.0) AND (#H_SP2 <= #MaxResSetp1) AND (#H_SP2 >= #MinResSetp1);
   #_w2 := (#H_SP2 <= #H_SPResonance1) AND #_w1;
   IF #_w2 THEN
       #H_SP2 := #MinResSetp1 - 0.5;
       #H_SetpntAllowed := FALSE;
   END_IF;
   #_w3 := (#H_SP2 > #H_SPResonance1) AND #_w1;
   IF #_w3 THEN
       #H_SP2 := #MaxResSetp1 + 0.5;
       #H_SetpntAllowed := FALSE;
   END_IF;
END_REGION

REGION Network 41: **** 5.2 - Equations - Flow Equations **** Check Setpoint 2 with Setpoint 2 Resonance
   // Check Setpoint 2 with Setpoint 2 Resonance 
   // Setpoint 2 is no longer allowed, calculate prefered allowed setpoint 2
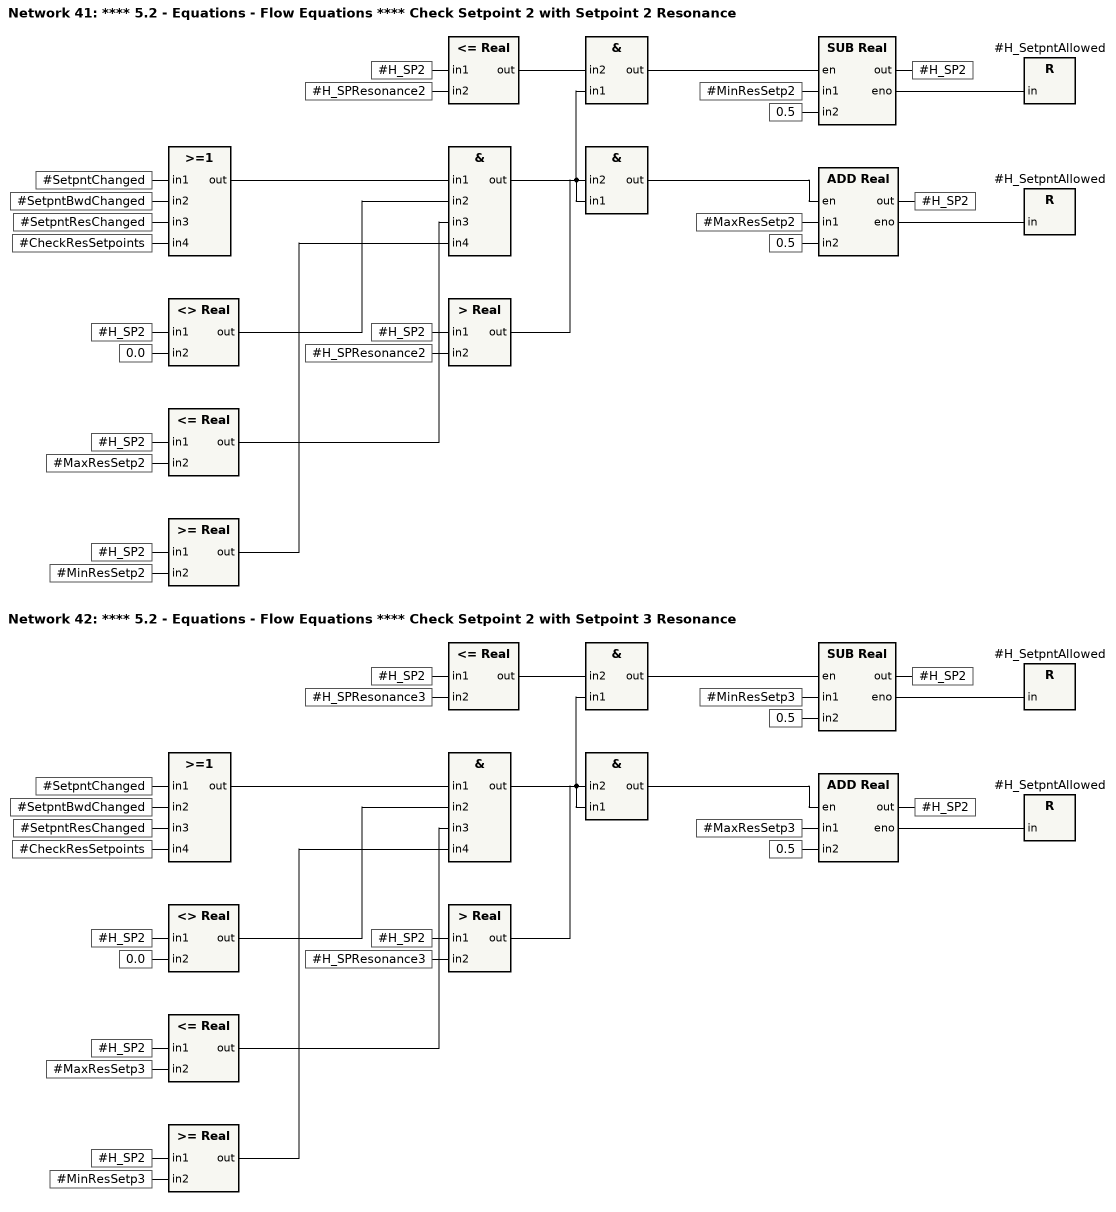
   // ENO of a box is taken as its EN; it also drops when the box reports an error
   #_w1 := (#SetpntChanged OR #SetpntBwdChanged OR #SetpntResChanged OR #CheckResSetpoints) AND (#H_SP2 <> 0.0) AND (#H_SP2 <= #MaxResSetp2) AND (#H_SP2 >= #MinResSetp2);
   #_w2 := (#H_SP2 <= #H_SPResonance2) AND #_w1;
   IF #_w2 THEN
       #H_SP2 := #MinResSetp2 - 0.5;
       #H_SetpntAllowed := FALSE;
   END_IF;
   #_w3 := (#H_SP2 > #H_SPResonance2) AND #_w1;
   IF #_w3 THEN
       #H_SP2 := #MaxResSetp2 + 0.5;
       #H_SetpntAllowed := FALSE;
   END_IF;
END_REGION

REGION Network 42: **** 5.2 - Equations - Flow Equations **** Check Setpoint 2 with Setpoint 3 Resonance
   // Check Setpoint 2 with Setpoint 3 Resonance 
   // Setpoint 2 is no longer allowed, calculate prefered allowed setpoint 2
   // ENO of a box is taken as its EN; it also drops when the box reports an error
   #_w1 := (#SetpntChanged OR #SetpntBwdChanged OR #SetpntResChanged OR #CheckResSetpoints) AND (#H_SP2 <> 0.0) AND (#H_SP2 <= #MaxResSetp3) AND (#H_SP2 >= #MinResSetp3);
   #_w2 := (#H_SP2 <= #H_SPResonance3) AND #_w1;
   IF #_w2 THEN
       #H_SP2 := #MinResSetp3 - 0.5;
       #H_SetpntAllowed := FALSE;
   END_IF;
   #_w3 := (#H_SP2 > #H_SPResonance3) AND #_w1;
   IF #_w3 THEN
       #H_SP2 := #MaxResSetp3 + 0.5;
       #H_SetpntAllowed := FALSE;
   END_IF;
END_REGION

REGION Network 43: **** 5.2 - Equations - Flow Equations **** Check Setpoint 2 with Setpoint 4 Resonance
   // Check Setpoint 2 with Setpoint 4 Resonance 
   // Setpoint 2 is no longer allowed, calculate prefered allowed setpoint 2
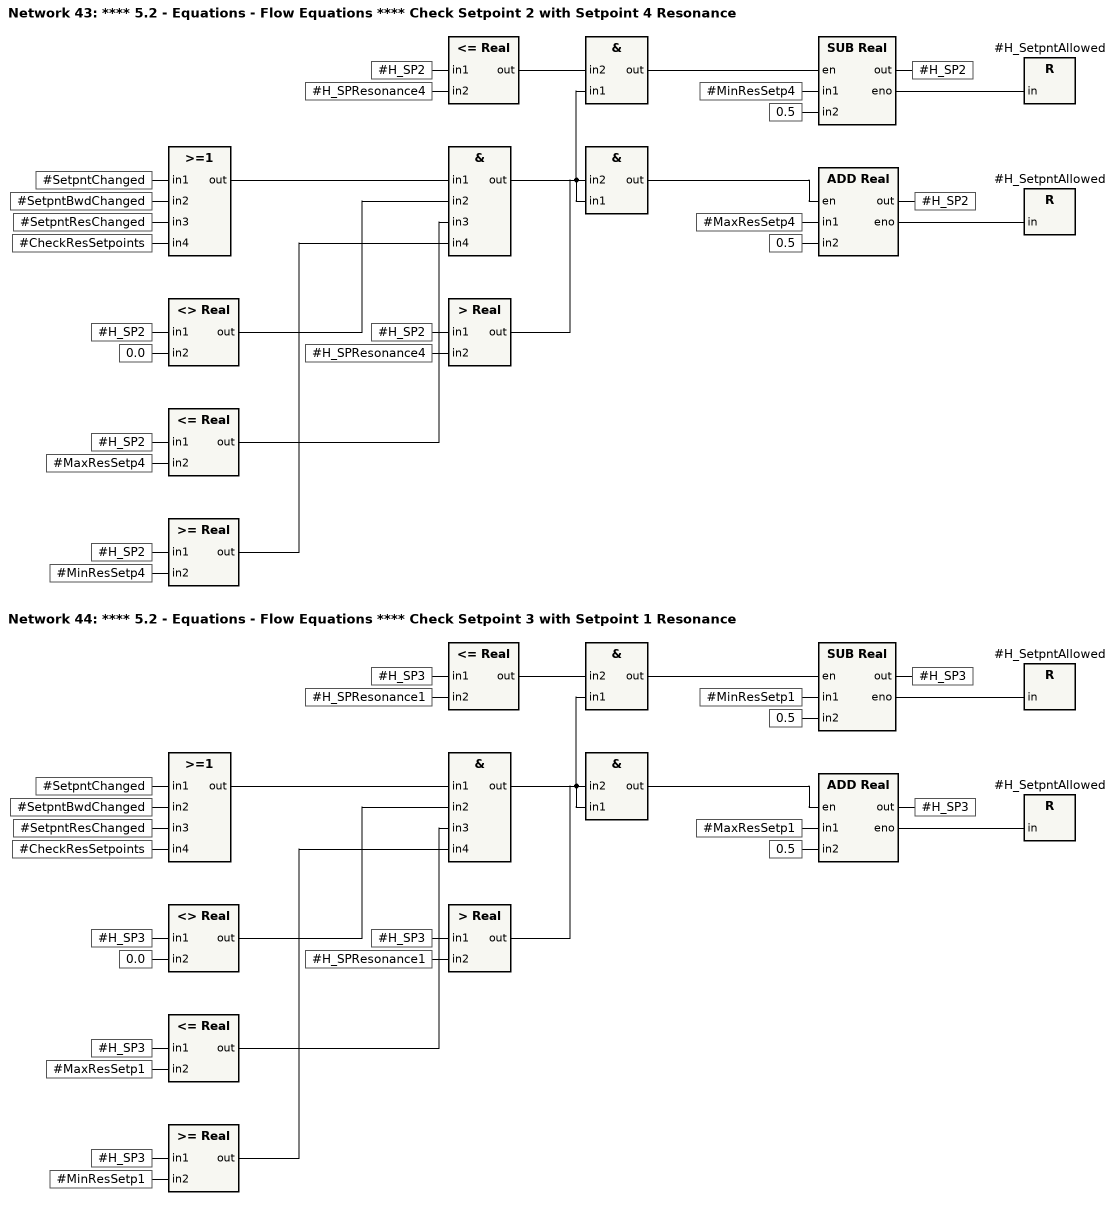
   // ENO of a box is taken as its EN; it also drops when the box reports an error
   #_w1 := (#SetpntChanged OR #SetpntBwdChanged OR #SetpntResChanged OR #CheckResSetpoints) AND (#H_SP2 <> 0.0) AND (#H_SP2 <= #MaxResSetp4) AND (#H_SP2 >= #MinResSetp4);
   #_w2 := (#H_SP2 <= #H_SPResonance4) AND #_w1;
   IF #_w2 THEN
       #H_SP2 := #MinResSetp4 - 0.5;
       #H_SetpntAllowed := FALSE;
   END_IF;
   #_w3 := (#H_SP2 > #H_SPResonance4) AND #_w1;
   IF #_w3 THEN
       #H_SP2 := #MaxResSetp4 + 0.5;
       #H_SetpntAllowed := FALSE;
   END_IF;
END_REGION

REGION Network 44: **** 5.2 - Equations - Flow Equations **** Check Setpoint 3 with Setpoint 1 Resonance
   // Check Setpoint 3 with Setpoint 1 Resonance 
   // Setpoint 3 is no longer allowed, calculate prefered allowed setpoint 3
   // ENO of a box is taken as its EN; it also drops when the box reports an error
   #_w1 := (#SetpntChanged OR #SetpntBwdChanged OR #SetpntResChanged OR #CheckResSetpoints) AND (#H_SP3 <> 0.0) AND (#H_SP3 <= #MaxResSetp1) AND (#H_SP3 >= #MinResSetp1);
   #_w2 := (#H_SP3 <= #H_SPResonance1) AND #_w1;
   IF #_w2 THEN
       #H_SP3 := #MinResSetp1 - 0.5;
       #H_SetpntAllowed := FALSE;
   END_IF;
   #_w3 := (#H_SP3 > #H_SPResonance1) AND #_w1;
   IF #_w3 THEN
       #H_SP3 := #MaxResSetp1 + 0.5;
       #H_SetpntAllowed := FALSE;
   END_IF;
END_REGION

REGION Network 45: **** 5.2 - Equations - Flow Equations **** Check Setpoint 3 with Setpoint 2 Resonance
   // Check Setpoint 3 with Setpoint 2 Resonance 
   // Setpoint 3 is no longer allowed, calculate prefered allowed setpoint 3
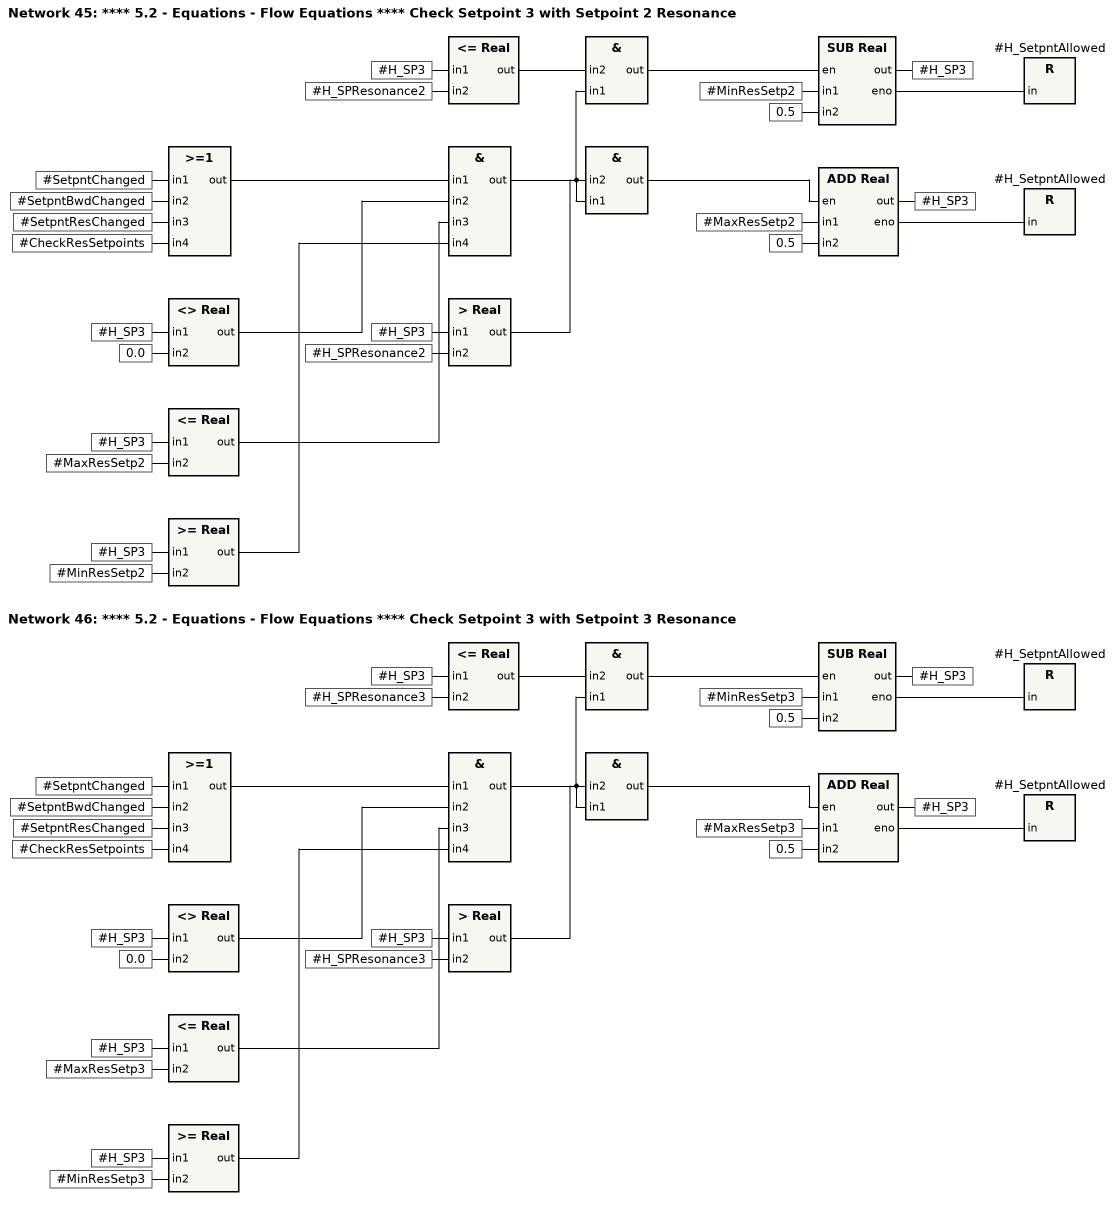
   // ENO of a box is taken as its EN; it also drops when the box reports an error
   #_w1 := (#SetpntChanged OR #SetpntBwdChanged OR #SetpntResChanged OR #CheckResSetpoints) AND (#H_SP3 <> 0.0) AND (#H_SP3 <= #MaxResSetp2) AND (#H_SP3 >= #MinResSetp2);
   #_w2 := (#H_SP3 <= #H_SPResonance2) AND #_w1;
   IF #_w2 THEN
       #H_SP3 := #MinResSetp2 - 0.5;
       #H_SetpntAllowed := FALSE;
   END_IF;
   #_w3 := (#H_SP3 > #H_SPResonance2) AND #_w1;
   IF #_w3 THEN
       #H_SP3 := #MaxResSetp2 + 0.5;
       #H_SetpntAllowed := FALSE;
   END_IF;
END_REGION

REGION Network 46: **** 5.2 - Equations - Flow Equations **** Check Setpoint 3 with Setpoint 3 Resonance
   // Check Setpoint 3 with Setpoint 3 Resonance 
   // Setpoint 3 is no longer allowed, calculate prefered allowed setpoint 3
   // ENO of a box is taken as its EN; it also drops when the box reports an error
   #_w1 := (#SetpntChanged OR #SetpntBwdChanged OR #SetpntResChanged OR #CheckResSetpoints) AND (#H_SP3 <> 0.0) AND (#H_SP3 <= #MaxResSetp3) AND (#H_SP3 >= #MinResSetp3);
   #_w2 := (#H_SP3 <= #H_SPResonance3) AND #_w1;
   IF #_w2 THEN
       #H_SP3 := #MinResSetp3 - 0.5;
       #H_SetpntAllowed := FALSE;
   END_IF;
   #_w3 := (#H_SP3 > #H_SPResonance3) AND #_w1;
   IF #_w3 THEN
       #H_SP3 := #MaxResSetp3 + 0.5;
       #H_SetpntAllowed := FALSE;
   END_IF;
END_REGION

REGION Network 47: **** 5.2 - Equations - Flow Equations **** Check Setpoint 3 with Setpoint 4 Resonance
   // Check Setpoint 3 with Setpoint 4 Resonance 
   // Setpoint 3 is no longer allowed, calculate prefered allowed setpoint 3
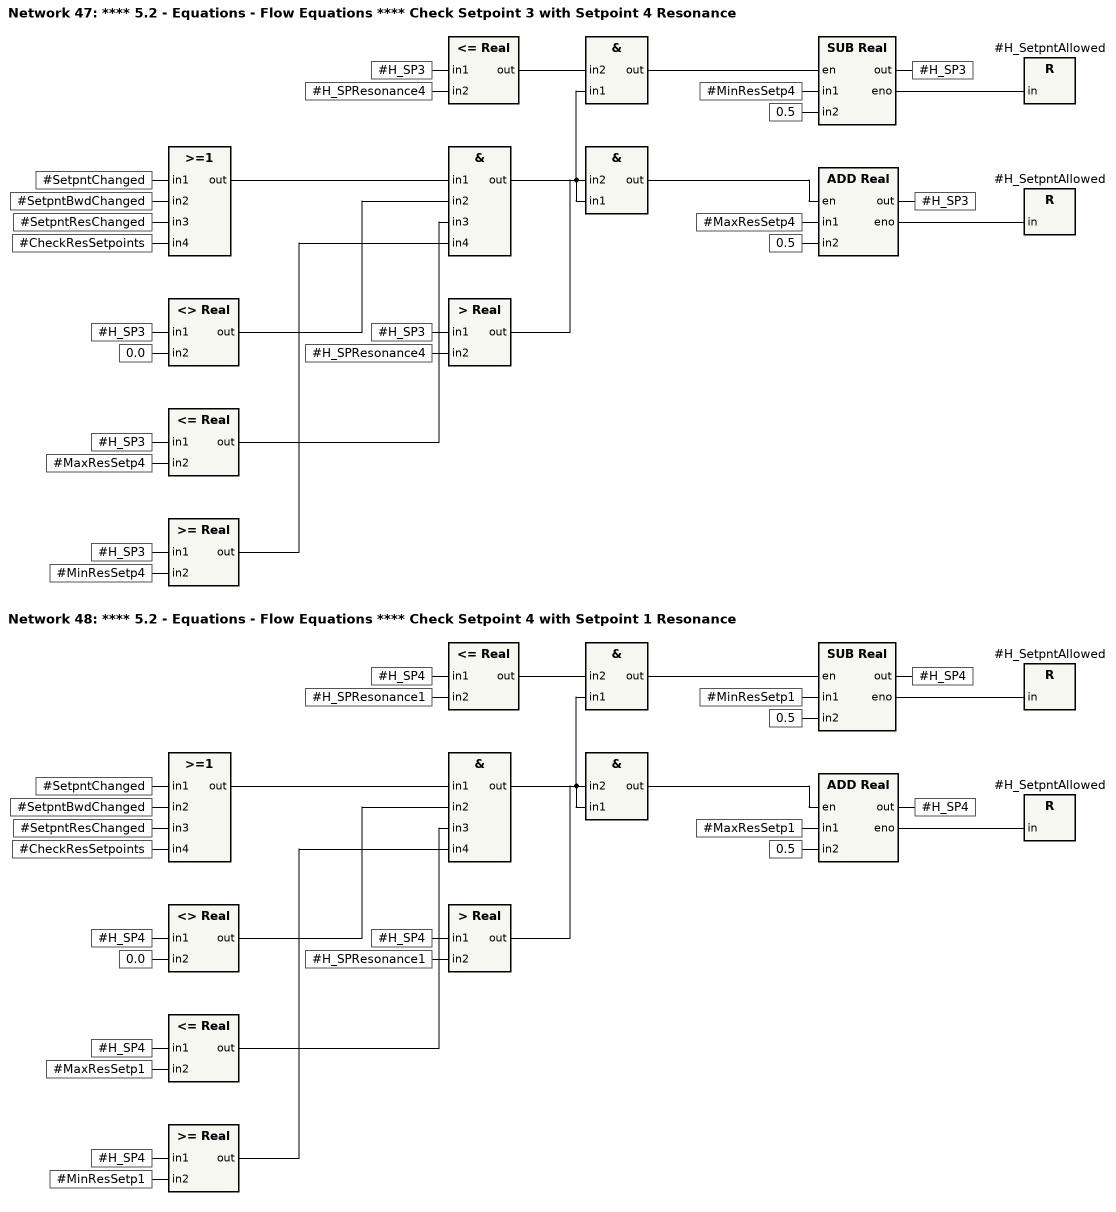
   // ENO of a box is taken as its EN; it also drops when the box reports an error
   #_w1 := (#SetpntChanged OR #SetpntBwdChanged OR #SetpntResChanged OR #CheckResSetpoints) AND (#H_SP3 <> 0.0) AND (#H_SP3 <= #MaxResSetp4) AND (#H_SP3 >= #MinResSetp4);
   #_w2 := (#H_SP3 <= #H_SPResonance4) AND #_w1;
   IF #_w2 THEN
       #H_SP3 := #MinResSetp4 - 0.5;
       #H_SetpntAllowed := FALSE;
   END_IF;
   #_w3 := (#H_SP3 > #H_SPResonance4) AND #_w1;
   IF #_w3 THEN
       #H_SP3 := #MaxResSetp4 + 0.5;
       #H_SetpntAllowed := FALSE;
   END_IF;
END_REGION

REGION Network 48: **** 5.2 - Equations - Flow Equations **** Check Setpoint 4 with Setpoint 1 Resonance
   // Check Setpoint 4 with Setpoint 1 Resonance 
   // Setpoint 4 is no longer allowed, calculate prefered allowed setpoint 4
   // ENO of a box is taken as its EN; it also drops when the box reports an error
   #_w1 := (#SetpntChanged OR #SetpntBwdChanged OR #SetpntResChanged OR #CheckResSetpoints) AND (#H_SP4 <> 0.0) AND (#H_SP4 <= #MaxResSetp1) AND (#H_SP4 >= #MinResSetp1);
   #_w2 := (#H_SP4 <= #H_SPResonance1) AND #_w1;
   IF #_w2 THEN
       #H_SP4 := #MinResSetp1 - 0.5;
       #H_SetpntAllowed := FALSE;
   END_IF;
   #_w3 := (#H_SP4 > #H_SPResonance1) AND #_w1;
   IF #_w3 THEN
       #H_SP4 := #MaxResSetp1 + 0.5;
       #H_SetpntAllowed := FALSE;
   END_IF;
END_REGION

REGION Network 49: **** 5.2 - Equations - Flow Equations **** Check Setpoint 4 with Setpoint 2 Resonance
   // Check Setpoint 4 with Setpoint 2 Resonance 
   // Setpoint 4 is no longer allowed, calculate prefered allowed setpoint 4
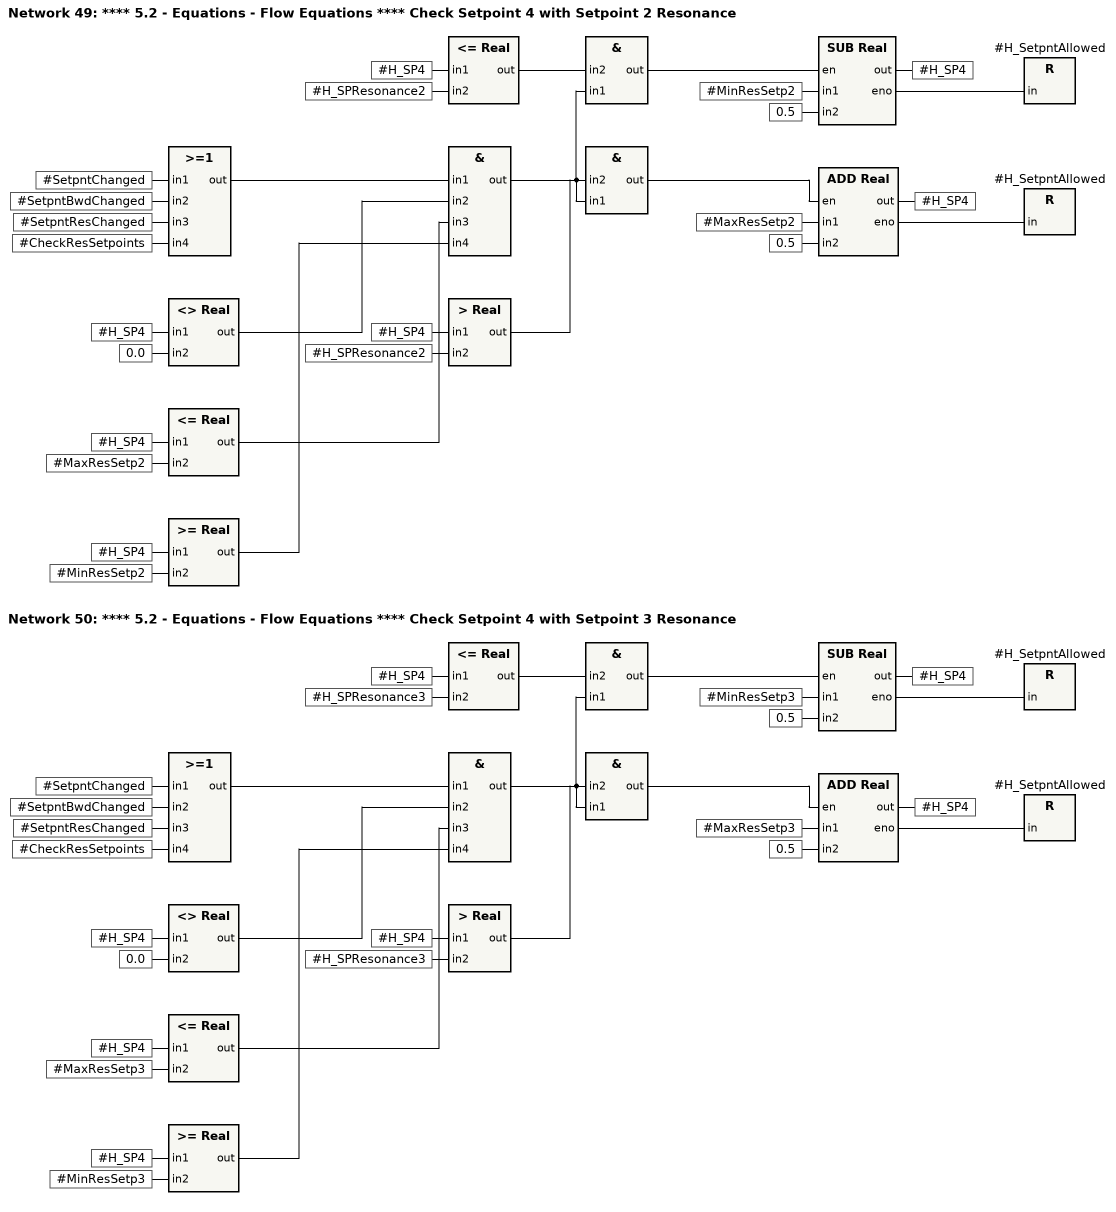
   // ENO of a box is taken as its EN; it also drops when the box reports an error
   #_w1 := (#SetpntChanged OR #SetpntBwdChanged OR #SetpntResChanged OR #CheckResSetpoints) AND (#H_SP4 <> 0.0) AND (#H_SP4 <= #MaxResSetp2) AND (#H_SP4 >= #MinResSetp2);
   #_w2 := (#H_SP4 <= #H_SPResonance2) AND #_w1;
   IF #_w2 THEN
       #H_SP4 := #MinResSetp2 - 0.5;
       #H_SetpntAllowed := FALSE;
   END_IF;
   #_w3 := (#H_SP4 > #H_SPResonance2) AND #_w1;
   IF #_w3 THEN
       #H_SP4 := #MaxResSetp2 + 0.5;
       #H_SetpntAllowed := FALSE;
   END_IF;
END_REGION

REGION Network 50: **** 5.2 - Equations - Flow Equations **** Check Setpoint 4 with Setpoint 3 Resonance
   // Check Setpoint 4 with Setpoint 3 Resonance 
   // Setpoint 4 is no longer allowed, calculate prefered allowed setpoint 4
   // ENO of a box is taken as its EN; it also drops when the box reports an error
   #_w1 := (#SetpntChanged OR #SetpntBwdChanged OR #SetpntResChanged OR #CheckResSetpoints) AND (#H_SP4 <> 0.0) AND (#H_SP4 <= #MaxResSetp3) AND (#H_SP4 >= #MinResSetp3);
   #_w2 := (#H_SP4 <= #H_SPResonance3) AND #_w1;
   IF #_w2 THEN
       #H_SP4 := #MinResSetp3 - 0.5;
       #H_SetpntAllowed := FALSE;
   END_IF;
   #_w3 := (#H_SP4 > #H_SPResonance3) AND #_w1;
   IF #_w3 THEN
       #H_SP4 := #MaxResSetp3 + 0.5;
       #H_SetpntAllowed := FALSE;
   END_IF;
END_REGION

REGION Network 51: **** 5.2 - Equations - Flow Equations **** Check Setpoint 4 with Setpoint 4 Resonance
   // Check Setpoint 4 with Setpoint 4 Resonance 
   // Setpoint 4 is no longer allowed, calculate prefered allowed setpoint 4
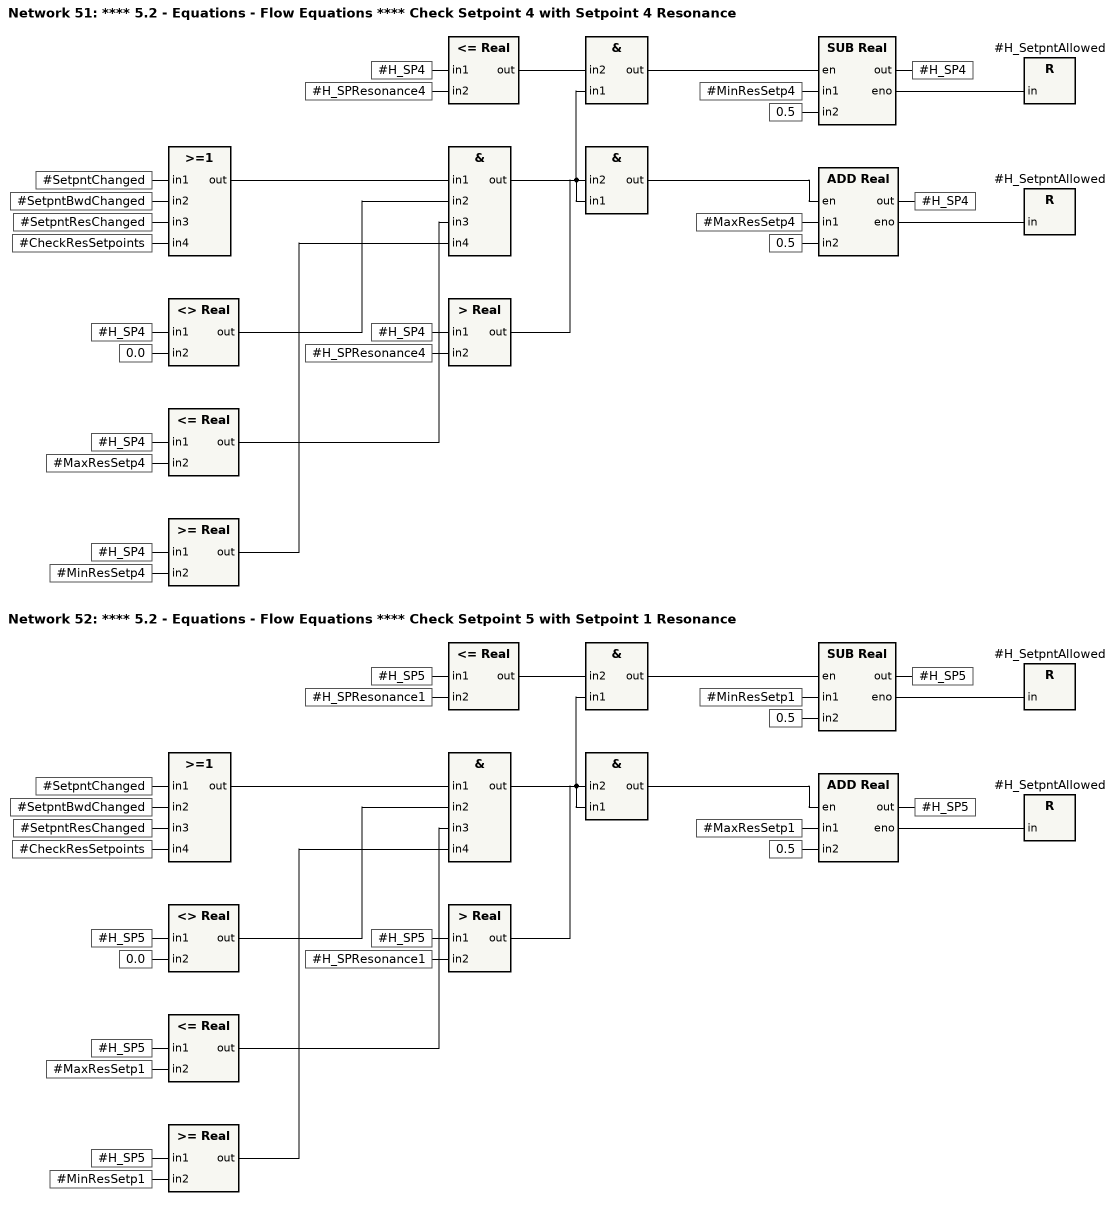
   // ENO of a box is taken as its EN; it also drops when the box reports an error
   #_w1 := (#SetpntChanged OR #SetpntBwdChanged OR #SetpntResChanged OR #CheckResSetpoints) AND (#H_SP4 <> 0.0) AND (#H_SP4 <= #MaxResSetp4) AND (#H_SP4 >= #MinResSetp4);
   #_w2 := (#H_SP4 <= #H_SPResonance4) AND #_w1;
   IF #_w2 THEN
       #H_SP4 := #MinResSetp4 - 0.5;
       #H_SetpntAllowed := FALSE;
   END_IF;
   #_w3 := (#H_SP4 > #H_SPResonance4) AND #_w1;
   IF #_w3 THEN
       #H_SP4 := #MaxResSetp4 + 0.5;
       #H_SetpntAllowed := FALSE;
   END_IF;
END_REGION

REGION Network 52: **** 5.2 - Equations - Flow Equations **** Check Setpoint 5 with Setpoint 1 Resonance
   // Check Setpoint 5 with Setpoint 1 Resonance 
   // Setpoint 5 is no longer allowed, calculate prefered allowed setpoint 5
   // ENO of a box is taken as its EN; it also drops when the box reports an error
   #_w1 := (#SetpntChanged OR #SetpntBwdChanged OR #SetpntResChanged OR #CheckResSetpoints) AND (#H_SP5 <> 0.0) AND (#H_SP5 <= #MaxResSetp1) AND (#H_SP5 >= #MinResSetp1);
   #_w2 := (#H_SP5 <= #H_SPResonance1) AND #_w1;
   IF #_w2 THEN
       #H_SP5 := #MinResSetp1 - 0.5;
       #H_SetpntAllowed := FALSE;
   END_IF;
   #_w3 := (#H_SP5 > #H_SPResonance1) AND #_w1;
   IF #_w3 THEN
       #H_SP5 := #MaxResSetp1 + 0.5;
       #H_SetpntAllowed := FALSE;
   END_IF;
END_REGION

REGION Network 53: **** 5.2 - Equations - Flow Equations ****Check Setpoint 5 with Setpoint 2 Resonance
   // Check Setpoint 5 with Setpoint 2 Resonance 
   // Setpoint 5 is no longer allowed, calculate prefered allowed setpoint 5
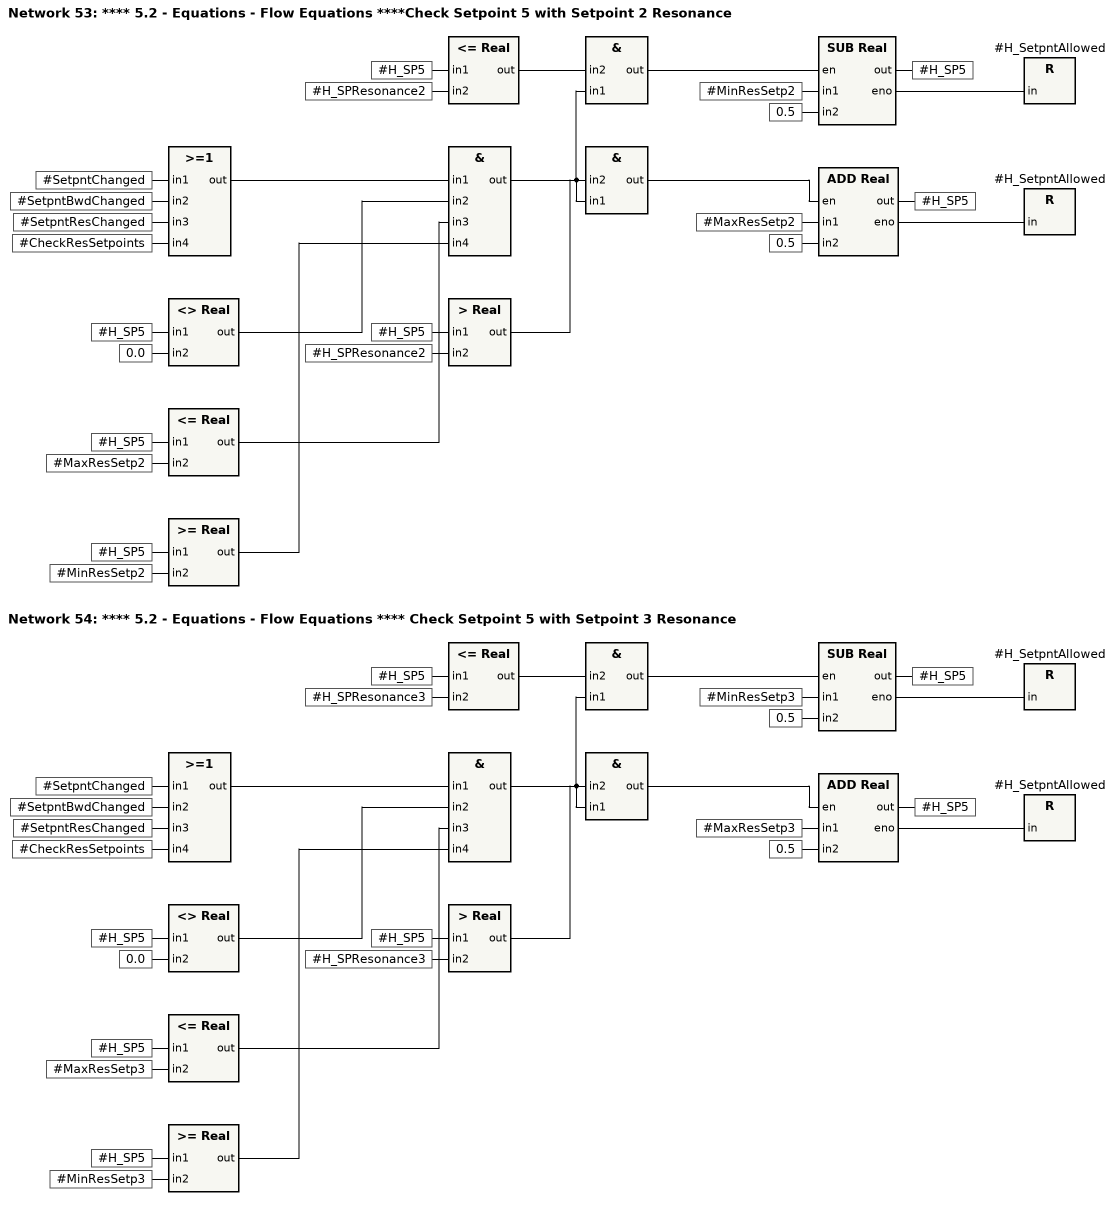
   // ENO of a box is taken as its EN; it also drops when the box reports an error
   #_w1 := (#SetpntChanged OR #SetpntBwdChanged OR #SetpntResChanged OR #CheckResSetpoints) AND (#H_SP5 <> 0.0) AND (#H_SP5 <= #MaxResSetp2) AND (#H_SP5 >= #MinResSetp2);
   #_w2 := (#H_SP5 <= #H_SPResonance2) AND #_w1;
   IF #_w2 THEN
       #H_SP5 := #MinResSetp2 - 0.5;
       #H_SetpntAllowed := FALSE;
   END_IF;
   #_w3 := (#H_SP5 > #H_SPResonance2) AND #_w1;
   IF #_w3 THEN
       #H_SP5 := #MaxResSetp2 + 0.5;
       #H_SetpntAllowed := FALSE;
   END_IF;
END_REGION

REGION Network 54: **** 5.2 - Equations - Flow Equations **** Check Setpoint 5 with Setpoint 3 Resonance
   // Check Setpoint 5 with Setpoint 3 Resonance 
   // Setpoint 5 is no longer allowed, calculate prefered allowed setpoint 5
   // ENO of a box is taken as its EN; it also drops when the box reports an error
   #_w1 := (#SetpntChanged OR #SetpntBwdChanged OR #SetpntResChanged OR #CheckResSetpoints) AND (#H_SP5 <> 0.0) AND (#H_SP5 <= #MaxResSetp3) AND (#H_SP5 >= #MinResSetp3);
   #_w2 := (#H_SP5 <= #H_SPResonance3) AND #_w1;
   IF #_w2 THEN
       #H_SP5 := #MinResSetp3 - 0.5;
       #H_SetpntAllowed := FALSE;
   END_IF;
   #_w3 := (#H_SP5 > #H_SPResonance3) AND #_w1;
   IF #_w3 THEN
       #H_SP5 := #MaxResSetp3 + 0.5;
       #H_SetpntAllowed := FALSE;
   END_IF;
END_REGION

REGION Network 55: **** 5.2 - Equations - Flow Equations **** Check Setpoint 5 with Setpoint 4 Resonance
   // Check Setpoint 5 with Setpoint 4 Resonance 
   // Setpoint 5 is no longer allowed, calculate prefered allowed setpoint 5
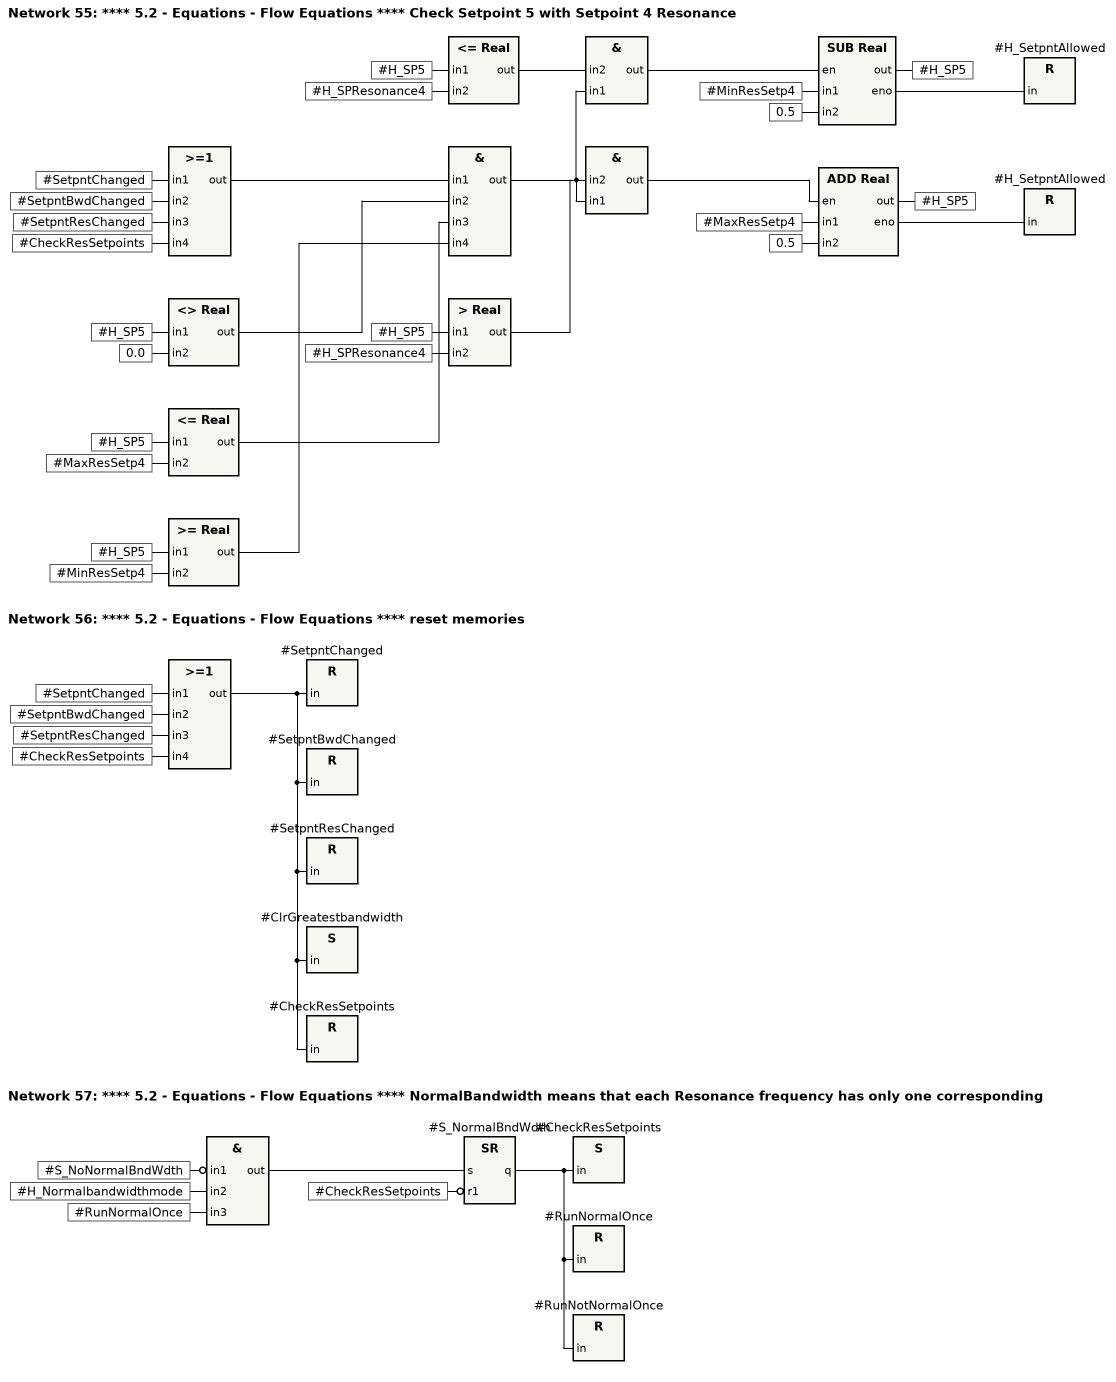
   // ENO of a box is taken as its EN; it also drops when the box reports an error
   #_w1 := (#SetpntChanged OR #SetpntBwdChanged OR #SetpntResChanged OR #CheckResSetpoints) AND (#H_SP5 <> 0.0) AND (#H_SP5 <= #MaxResSetp4) AND (#H_SP5 >= #MinResSetp4);
   #_w2 := (#H_SP5 <= #H_SPResonance4) AND #_w1;
   IF #_w2 THEN
       #H_SP5 := #MinResSetp4 - 0.5;
       #H_SetpntAllowed := FALSE;
   END_IF;
   #_w3 := (#H_SP5 > #H_SPResonance4) AND #_w1;
   IF #_w3 THEN
       #H_SP5 := #MaxResSetp4 + 0.5;
       #H_SetpntAllowed := FALSE;
   END_IF;
END_REGION

REGION Network 56: **** 5.2 - Equations - Flow Equations **** reset memories
   // reset memories
   #_w1 := #SetpntChanged OR #SetpntBwdChanged OR #SetpntResChanged OR #CheckResSetpoints;
   IF #_w1 THEN
       #SetpntChanged := FALSE;
       #SetpntBwdChanged := FALSE;
       #SetpntResChanged := FALSE;
       #ClrGreatestbandwidth := TRUE;
       #CheckResSetpoints := FALSE;
   END_IF;
END_REGION

REGION Network 57: **** 5.2 - Equations - Flow Equations **** NormalBandwidth means that each Resonance frequency has only one corresponding
   // NormalBandwidth means that each Resonance frequency has only one corresponding 
   // bandwidth
   IF NOT #S_NoNormalBndWdth AND #H_Normalbandwidthmode AND #RunNormalOnce THEN
       #S_NormalBndWdth := TRUE;   // SR flip-flop
   END_IF;
   IF NOT #CheckResSetpoints THEN #S_NormalBndWdth := FALSE; END_IF;
   IF #S_NormalBndWdth THEN
       #CheckResSetpoints := TRUE;
       #RunNormalOnce := FALSE;
       #RunNotNormalOnce := FALSE;
   END_IF;
END_REGION

REGION Network 58: **** 5.2 - Equations - Flow Equations **** Not NormalBandwidth means that each Resonance frequency works with the greatest
   // Not NormalBandwidth means that each Resonance frequency works with the greatest 
   // value of the 4 bandwidth's; it corresponds with the parametrizing of Danfoss 
   // frequency controller
   // bandwidth
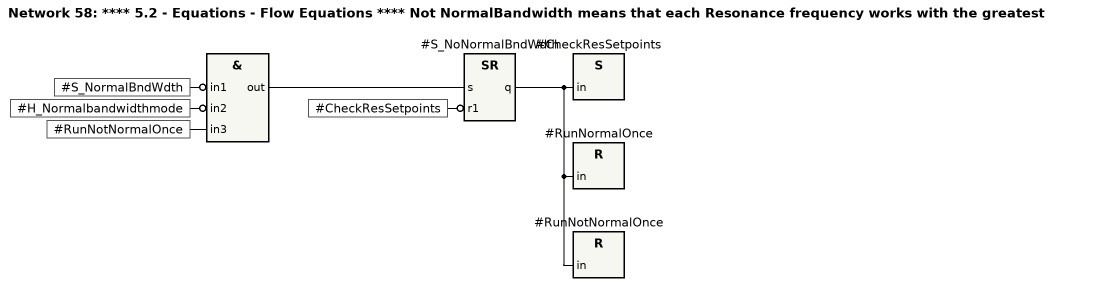
   IF NOT #S_NormalBndWdth AND NOT #H_Normalbandwidthmode AND #RunNotNormalOnce THEN
       #S_NoNormalBndWdth := TRUE;   // SR flip-flop
   END_IF;
   IF NOT #CheckResSetpoints THEN #S_NoNormalBndWdth := FALSE; END_IF;
   IF #S_NoNormalBndWdth THEN
       #CheckResSetpoints := TRUE;
       #RunNormalOnce := FALSE;
       #RunNotNormalOnce := FALSE;
   END_IF;
END_REGION
END_FUNCTION_BLOCK
